(*SOA 12.01.2023 {  *)
(* QVis page 141, Warm up *)
iIndexPage:=141;
iPageNumber:=iPageNumber+1;
T_Visu.T_PageIndex[iIndexPage].iIndexConfigPage:=iPageNumber;
ptrConfigPage:=ADR(T_Visu.T_ConfigPage[T_Visu.T_PageIndex[iIndexPage].iIndexConfigPage]);
ptrConfigPage^.sName:='Warm up';
ptrConfigPage^.wMaskBtPanelLeft:=16#1F;
ptrConfigPage^.wMaskBtPanelRight:=16#60;
ptrConfigPage^.wMaskFunctionPanel:=16#31;
(* Navigation panel restriction *)
ptrConfigPage^.wMaskTouchScreenNavPanel:=16#3F;
(* Active machine movement mask *)
ptrConfigPage^.wMaskActiveMachineBtPanelLeft:=16#0;
ptrConfigPage^.wMaskActiveMachineBtPanelRight:=16#0;
ptrConfigPage^.wMaskActiveMachineFunctionPanel:=16#0;
ptrConfigPage^.wMaskActiveMachineNavPanel:=16#3F;
(* Button edge action *)
ptrConfigPage^.aiRTrigActionPanelRight[1]:=10140;
ptrConfigPage^.aiRTrigActionPanelRight[2]:=10141;
ptrConfigPage^.aiRTrigActionPanelRight[3]:=0;
ptrConfigPage^.aiRTrigActionPanelRight[4]:=0;
ptrConfigPage^.aiRTrigActionPanelRight[5]:=0;
ptrConfigPage^.aiFTrigActionPanelRight[1]:=0;
ptrConfigPage^.aiFTrigActionPanelRight[2]:=0;
ptrConfigPage^.aiFTrigActionPanelRight[3]:=0;
ptrConfigPage^.aiFTrigActionPanelRight[4]:=0;
ptrConfigPage^.aiFTrigActionPanelRight[5]:=0;
ptrConfigPage^.aiDelayActionPanelRight[1]:=0;
ptrConfigPage^.aiDelayActionPanelRight[2]:=0;
ptrConfigPage^.aiDelayActionPanelRight[3]:=0;
ptrConfigPage^.aiDelayActionPanelRight[4]:=0;
ptrConfigPage^.aiDelayActionPanelRight[5]:=0;
ptrConfigPage^.aiRTrigActionFunctionPanel[1]:=173;
ptrConfigPage^.aiRTrigActionFunctionPanel[2]:=0;
ptrConfigPage^.aiRTrigActionFunctionPanel[3]:=0;
ptrConfigPage^.aiRTrigActionFunctionPanel[4]:=0;
ptrConfigPage^.aiRTrigActionFunctionPanel[5]:=175;
ptrConfigPage^.aiRTrigActionFunctionPanel[6]:= 1005; (*Vorher: 171*)
ptrConfigPage^.aiRTrigActionFunctionPanel[7]:=0;
ptrConfigPage^.aiRTrigActionFunctionPanel[8]:=0;
ptrConfigPage^.aiRTrigActionFunctionPanel[9]:=0;
ptrConfigPage^.aiRTrigActionFunctionPanel[10]:=0;
ptrConfigPage^.aiRTrigActionFunctionPanel[11]:=0;
ptrConfigPage^.aiRTrigActionFunctionPanel[12]:=0;
ptrConfigPage^.aiFTrigActionTouchScreenNavPanel[1]:=10110;
ptrConfigPage^.aiFTrigActionTouchScreenNavPanel[2]:=10120;
ptrConfigPage^.aiFTrigActionTouchScreenNavPanel[3]:=10130;
ptrConfigPage^.aiFTrigActionTouchScreenNavPanel[4]:=10140;
ptrConfigPage^.aiFTrigActionTouchScreenNavPanel[5]:=10150;
ptrConfigPage^.aiFTrigActionTouchScreenNavPanel[6]:=10160;
ptrConfigPage^.xMaskBtStart:=FALSE;
ptrConfigPage^.xMaskBtStop:=TRUE;
(*SOA 12.01.2023 }  *)

(* QVis page 150, Configuration *)
iIndexPage:=150;
iPageNumber:=iPageNumber+1;
T_Visu.T_PageIndex[iIndexPage].iIndexConfigPage:=iPageNumber;
ptrConfigPage:=ADR(T_Visu.T_ConfigPage[T_Visu.T_PageIndex[iIndexPage].iIndexConfigPage]);
ptrConfigPage^.sName:='Configuration';
ptrConfigPage^.wMaskBtPanelLeft:=16#1F;
ptrConfigPage^.wMaskBtPanelRight:=16#0;
ptrConfigPage^.wMaskFunctionPanel:=16#0;
(* Navigation panel restriction *)
ptrConfigPage^.wMaskTouchScreenNavPanel:=16#3F;
(* Active machine movement mask *)
ptrConfigPage^.wMaskActiveMachineBtPanelLeft:=16#0;
ptrConfigPage^.wMaskActiveMachineBtPanelRight:=16#0;
ptrConfigPage^.wMaskActiveMachineFunctionPanel:=16#0;
ptrConfigPage^.wMaskActiveMachineNavPanel:=16#3F;
(* Button edge action *)
ptrConfigPage^.aiRTrigActionPanelRight[1]:=0;
ptrConfigPage^.aiRTrigActionPanelRight[2]:=0;
ptrConfigPage^.aiRTrigActionPanelRight[3]:=0;
ptrConfigPage^.aiRTrigActionPanelRight[4]:=0;
ptrConfigPage^.aiRTrigActionPanelRight[5]:=0;
ptrConfigPage^.aiFTrigActionPanelRight[1]:=0;
ptrConfigPage^.aiFTrigActionPanelRight[2]:=0;
ptrConfigPage^.aiFTrigActionPanelRight[3]:=0;
ptrConfigPage^.aiFTrigActionPanelRight[4]:=0;
ptrConfigPage^.aiFTrigActionPanelRight[5]:=0;
ptrConfigPage^.aiDelayActionPanelRight[1]:=0;
ptrConfigPage^.aiDelayActionPanelRight[2]:=0;
ptrConfigPage^.aiDelayActionPanelRight[3]:=0;
ptrConfigPage^.aiDelayActionPanelRight[4]:=0;
ptrConfigPage^.aiDelayActionPanelRight[5]:=0;
ptrConfigPage^.aiRTrigActionFunctionPanel[1]:=0;
ptrConfigPage^.aiRTrigActionFunctionPanel[2]:=0;
ptrConfigPage^.aiRTrigActionFunctionPanel[3]:=0;
ptrConfigPage^.aiRTrigActionFunctionPanel[4]:=0;
ptrConfigPage^.aiRTrigActionFunctionPanel[5]:=0;
ptrConfigPage^.aiRTrigActionFunctionPanel[6]:=0;
ptrConfigPage^.aiRTrigActionFunctionPanel[7]:=0;
ptrConfigPage^.aiRTrigActionFunctionPanel[8]:=0;
ptrConfigPage^.aiRTrigActionFunctionPanel[9]:=0;
ptrConfigPage^.aiRTrigActionFunctionPanel[10]:=0;
ptrConfigPage^.aiRTrigActionFunctionPanel[11]:=0;
ptrConfigPage^.aiRTrigActionFunctionPanel[12]:=0;
ptrConfigPage^.aiFTrigActionTouchScreenNavPanel[1]:=10110;
ptrConfigPage^.aiFTrigActionTouchScreenNavPanel[2]:=10120;
ptrConfigPage^.aiFTrigActionTouchScreenNavPanel[3]:=10130;
ptrConfigPage^.aiFTrigActionTouchScreenNavPanel[4]:=10140;
ptrConfigPage^.aiFTrigActionTouchScreenNavPanel[5]:=10150;
ptrConfigPage^.aiFTrigActionTouchScreenNavPanel[6]:=10160;
ptrConfigPage^.xMaskBtStart:=FALSE;
ptrConfigPage^.xMaskBtStop:=TRUE;

(* QVis page 160, Error List *)
iIndexPage:=160;
iPageNumber:=iPageNumber+1;
T_Visu.T_PageIndex[iIndexPage].iIndexConfigPage:=iPageNumber;
ptrConfigPage:=ADR(T_Visu.T_ConfigPage[T_Visu.T_PageIndex[iIndexPage].iIndexConfigPage]);
ptrConfigPage^.sName:='Error List';
ptrConfigPage^.wMaskBtPanelLeft:=16#1F;
ptrConfigPage^.wMaskBtPanelRight:=16#60;
ptrConfigPage^.wMaskFunctionPanel:=16#0;
(* Navigation panel restriction *)
ptrConfigPage^.wMaskTouchScreenNavPanel:=16#3F;
(* Active machine movement mask *)
ptrConfigPage^.wMaskActiveMachineBtPanelLeft:=16#0;
ptrConfigPage^.wMaskActiveMachineBtPanelRight:=16#60;
ptrConfigPage^.wMaskActiveMachineFunctionPanel:=16#0;
ptrConfigPage^.wMaskActiveMachineNavPanel:=16#3F;
(* Button edge action *)
ptrConfigPage^.aiRTrigActionPanelRight[1]:=99;
ptrConfigPage^.aiRTrigActionPanelRight[2]:=20;
ptrConfigPage^.aiRTrigActionPanelRight[3]:=0;
ptrConfigPage^.aiRTrigActionPanelRight[4]:=0;
ptrConfigPage^.aiRTrigActionPanelRight[5]:=0;
ptrConfigPage^.aiFTrigActionPanelRight[1]:=0;
ptrConfigPage^.aiFTrigActionPanelRight[2]:=0;
ptrConfigPage^.aiFTrigActionPanelRight[3]:=0;
ptrConfigPage^.aiFTrigActionPanelRight[4]:=0;
ptrConfigPage^.aiFTrigActionPanelRight[5]:=0;
ptrConfigPage^.aiDelayActionPanelRight[1]:=0;
ptrConfigPage^.aiDelayActionPanelRight[2]:=0;
ptrConfigPage^.aiDelayActionPanelRight[3]:=0;
ptrConfigPage^.aiDelayActionPanelRight[4]:=0;
ptrConfigPage^.aiDelayActionPanelRight[5]:=0;
ptrConfigPage^.aiRTrigActionFunctionPanel[1]:=0;
ptrConfigPage^.aiRTrigActionFunctionPanel[2]:=0;
ptrConfigPage^.aiRTrigActionFunctionPanel[3]:=0;
ptrConfigPage^.aiRTrigActionFunctionPanel[4]:=0;
ptrConfigPage^.aiRTrigActionFunctionPanel[5]:=0;
ptrConfigPage^.aiRTrigActionFunctionPanel[6]:=0;
ptrConfigPage^.aiRTrigActionFunctionPanel[7]:=0;
ptrConfigPage^.aiRTrigActionFunctionPanel[8]:=0;
ptrConfigPage^.aiRTrigActionFunctionPanel[9]:=0;
ptrConfigPage^.aiRTrigActionFunctionPanel[10]:=0;
ptrConfigPage^.aiRTrigActionFunctionPanel[11]:=0;
ptrConfigPage^.aiRTrigActionFunctionPanel[12]:=0;
ptrConfigPage^.aiFTrigActionTouchScreenNavPanel[1]:=10110;
ptrConfigPage^.aiFTrigActionTouchScreenNavPanel[2]:=10120;
ptrConfigPage^.aiFTrigActionTouchScreenNavPanel[3]:=10130;
ptrConfigPage^.aiFTrigActionTouchScreenNavPanel[4]:=10140;
ptrConfigPage^.aiFTrigActionTouchScreenNavPanel[5]:=10150;
ptrConfigPage^.aiFTrigActionTouchScreenNavPanel[6]:=10160;
ptrConfigPage^.xMaskBtStart:=FALSE;
ptrConfigPage^.xMaskBtStop:=TRUE;

(* QVis page 170, Parameter General *)
iIndexPage:=170;
iPageNumber:=iPageNumber+1;
T_Visu.T_PageIndex[iIndexPage].iIndexConfigPage:=iPageNumber;
ptrConfigPage:=ADR(T_Visu.T_ConfigPage[T_Visu.T_PageIndex[iIndexPage].iIndexConfigPage]);
ptrConfigPage^.sName:='Parameter General';
ptrConfigPage^.wMaskBtPanelLeft:=16#1F;
ptrConfigPage^.wMaskBtPanelRight:=16#200;
ptrConfigPage^.wMaskFunctionPanel:=16#0;
(* Navigation panel restriction *)
ptrConfigPage^.wMaskTouchScreenNavPanel:=16#3F;
(* Active machine movement mask *)
ptrConfigPage^.wMaskActiveMachineBtPanelLeft:=16#0;
ptrConfigPage^.wMaskActiveMachineBtPanelRight:=16#0;
ptrConfigPage^.wMaskActiveMachineFunctionPanel:=16#0;
ptrConfigPage^.wMaskActiveMachineNavPanel:=16#3F;
(* Button edge action *)
ptrConfigPage^.aiRTrigActionPanelRight[1]:=0;
ptrConfigPage^.aiRTrigActionPanelRight[2]:=0;
ptrConfigPage^.aiRTrigActionPanelRight[3]:=0;
ptrConfigPage^.aiRTrigActionPanelRight[4]:=0;
ptrConfigPage^.aiRTrigActionPanelRight[5]:=1006;
ptrConfigPage^.aiFTrigActionPanelRight[1]:=0;
ptrConfigPage^.aiFTrigActionPanelRight[2]:=0;
ptrConfigPage^.aiFTrigActionPanelRight[3]:=0;
ptrConfigPage^.aiFTrigActionPanelRight[4]:=0;
ptrConfigPage^.aiFTrigActionPanelRight[5]:=0;
ptrConfigPage^.aiDelayActionPanelRight[1]:=0;
ptrConfigPage^.aiDelayActionPanelRight[2]:=0;
ptrConfigPage^.aiDelayActionPanelRight[3]:=0;
ptrConfigPage^.aiDelayActionPanelRight[4]:=0;
ptrConfigPage^.aiDelayActionPanelRight[5]:=0;
ptrConfigPage^.aiRTrigActionFunctionPanel[1]:=0;
ptrConfigPage^.aiRTrigActionFunctionPanel[2]:=0;
ptrConfigPage^.aiRTrigActionFunctionPanel[3]:=0;
ptrConfigPage^.aiRTrigActionFunctionPanel[4]:=0;
ptrConfigPage^.aiRTrigActionFunctionPanel[5]:=0;
ptrConfigPage^.aiRTrigActionFunctionPanel[6]:=0;
ptrConfigPage^.aiRTrigActionFunctionPanel[7]:=0;
ptrConfigPage^.aiRTrigActionFunctionPanel[8]:=0;
ptrConfigPage^.aiRTrigActionFunctionPanel[9]:=0;
ptrConfigPage^.aiRTrigActionFunctionPanel[10]:=0;
ptrConfigPage^.aiRTrigActionFunctionPanel[11]:=0;
ptrConfigPage^.aiRTrigActionFunctionPanel[12]:=0;
ptrConfigPage^.aiFTrigActionTouchScreenNavPanel[1]:=10110;
ptrConfigPage^.aiFTrigActionTouchScreenNavPanel[2]:=10120;
ptrConfigPage^.aiFTrigActionTouchScreenNavPanel[3]:=10130;
ptrConfigPage^.aiFTrigActionTouchScreenNavPanel[4]:=10140;
ptrConfigPage^.aiFTrigActionTouchScreenNavPanel[5]:=10150;
ptrConfigPage^.aiFTrigActionTouchScreenNavPanel[6]:=10160;
ptrConfigPage^.xMaskBtStart:=FALSE;
ptrConfigPage^.xMaskBtStop:=TRUE;

(* QVis page 210, Teach-in Tool Rotation *)
iIndexPage:=210;
iPageNumber:=iPageNumber+1;
T_Visu.T_PageIndex[iIndexPage].iIndexConfigPage:=iPageNumber;
ptrConfigPage:=ADR(T_Visu.T_ConfigPage[T_Visu.T_PageIndex[iIndexPage].iIndexConfigPage]);
ptrConfigPage^.sName:='Teach-in Tool Rotation';
ptrConfigPage^.wMaskBtPanelLeft:=16#1F;
ptrConfigPage^.wMaskBtPanelRight:=16#1E0;
ptrConfigPage^.wMaskFunctionPanel:=16#F;
(* Navigation panel restriction *)
ptrConfigPage^.wMaskTouchScreenNavPanel:=16#27;
(* Active machine movement mask *)
ptrConfigPage^.wMaskActiveMachineBtPanelLeft:=16#0;
ptrConfigPage^.wMaskActiveMachineBtPanelRight:=16#0;
ptrConfigPage^.wMaskActiveMachineFunctionPanel:=16#0;
ptrConfigPage^.wMaskActiveMachineNavPanel:=16#27;
(* Button edge action *)
ptrConfigPage^.aiRTrigActionPanelRight[1]:=312;
ptrConfigPage^.aiRTrigActionPanelRight[2]:=310;
ptrConfigPage^.aiRTrigActionPanelRight[3]:=316;
ptrConfigPage^.aiRTrigActionPanelRight[4]:=314;
ptrConfigPage^.aiRTrigActionPanelRight[5]:=0;
ptrConfigPage^.aiFTrigActionPanelRight[1]:=0;
ptrConfigPage^.aiFTrigActionPanelRight[2]:=0;
ptrConfigPage^.aiFTrigActionPanelRight[3]:=301;
ptrConfigPage^.aiFTrigActionPanelRight[4]:=301;
ptrConfigPage^.aiFTrigActionPanelRight[5]:=0;
ptrConfigPage^.aiDelayActionPanelRight[1]:=0;
ptrConfigPage^.aiDelayActionPanelRight[2]:=0;
ptrConfigPage^.aiDelayActionPanelRight[3]:=0;
ptrConfigPage^.aiDelayActionPanelRight[4]:=0;
ptrConfigPage^.aiDelayActionPanelRight[5]:=0;
ptrConfigPage^.aiRTrigActionFunctionPanel[1]:=322;
ptrConfigPage^.aiRTrigActionFunctionPanel[2]:=323;
ptrConfigPage^.aiRTrigActionFunctionPanel[3]:=321;
ptrConfigPage^.aiRTrigActionFunctionPanel[4]:=320;
ptrConfigPage^.aiRTrigActionFunctionPanel[5]:=0;
ptrConfigPage^.aiRTrigActionFunctionPanel[6]:=0;
ptrConfigPage^.aiRTrigActionFunctionPanel[7]:=0;
ptrConfigPage^.aiRTrigActionFunctionPanel[8]:=0;
ptrConfigPage^.aiRTrigActionFunctionPanel[9]:=0;
ptrConfigPage^.aiRTrigActionFunctionPanel[10]:=0;
ptrConfigPage^.aiRTrigActionFunctionPanel[11]:=0;
ptrConfigPage^.aiRTrigActionFunctionPanel[12]:=0;
ptrConfigPage^.aiFTrigActionTouchScreenNavPanel[1]:=10210;
ptrConfigPage^.aiFTrigActionTouchScreenNavPanel[2]:=10220;
ptrConfigPage^.aiFTrigActionTouchScreenNavPanel[3]:=10230;
ptrConfigPage^.aiFTrigActionTouchScreenNavPanel[4]:=0;
ptrConfigPage^.aiFTrigActionTouchScreenNavPanel[5]:=0;
ptrConfigPage^.aiFTrigActionTouchScreenNavPanel[6]:=10260;
ptrConfigPage^.xMaskBtStart:=TRUE;
ptrConfigPage^.xMaskBtStop:=TRUE;

(* QVis page 220, Tool Torque *)
iIndexPage:=220;
iPageNumber:=iPageNumber+1;
T_Visu.T_PageIndex[iIndexPage].iIndexConfigPage:=iPageNumber;
ptrConfigPage:=ADR(T_Visu.T_ConfigPage[T_Visu.T_PageIndex[iIndexPage].iIndexConfigPage]);
ptrConfigPage^.sName:='Tool Torque';
ptrConfigPage^.wMaskBtPanelLeft:=16#1F;
ptrConfigPage^.wMaskBtPanelRight:=16#0;
ptrConfigPage^.wMaskFunctionPanel:=16#DF;
(* Navigation panel restriction *)
ptrConfigPage^.wMaskTouchScreenNavPanel:=16#27;
(* Active machine movement mask *)
ptrConfigPage^.wMaskActiveMachineBtPanelLeft:=16#0;
ptrConfigPage^.wMaskActiveMachineBtPanelRight:=16#0;
ptrConfigPage^.wMaskActiveMachineFunctionPanel:=16#DF;
ptrConfigPage^.wMaskActiveMachineNavPanel:=16#27;
(* Button edge action *)
ptrConfigPage^.aiRTrigActionPanelRight[1]:=0;
ptrConfigPage^.aiRTrigActionPanelRight[2]:=0;
ptrConfigPage^.aiRTrigActionPanelRight[3]:=0;
ptrConfigPage^.aiRTrigActionPanelRight[4]:=0;
ptrConfigPage^.aiRTrigActionPanelRight[5]:=0;
ptrConfigPage^.aiFTrigActionPanelRight[1]:=0;
ptrConfigPage^.aiFTrigActionPanelRight[2]:=0;
ptrConfigPage^.aiFTrigActionPanelRight[3]:=0;
ptrConfigPage^.aiFTrigActionPanelRight[4]:=0;
ptrConfigPage^.aiFTrigActionPanelRight[5]:=0;
ptrConfigPage^.aiDelayActionPanelRight[1]:=0;
ptrConfigPage^.aiDelayActionPanelRight[2]:=0;
ptrConfigPage^.aiDelayActionPanelRight[3]:=0;
ptrConfigPage^.aiDelayActionPanelRight[4]:=0;
ptrConfigPage^.aiDelayActionPanelRight[5]:=0;
ptrConfigPage^.aiRTrigActionFunctionPanel[1]:=502;
ptrConfigPage^.aiRTrigActionFunctionPanel[2]:=503;
ptrConfigPage^.aiRTrigActionFunctionPanel[3]:=501;
ptrConfigPage^.aiRTrigActionFunctionPanel[4]:=130;
ptrConfigPage^.aiRTrigActionFunctionPanel[5]:=131;
ptrConfigPage^.aiRTrigActionFunctionPanel[6]:=0;
ptrConfigPage^.aiRTrigActionFunctionPanel[7]:=504;
ptrConfigPage^.aiRTrigActionFunctionPanel[8]:=505;
ptrConfigPage^.aiRTrigActionFunctionPanel[9]:=0;
ptrConfigPage^.aiRTrigActionFunctionPanel[10]:=0;
ptrConfigPage^.aiRTrigActionFunctionPanel[11]:=0;
ptrConfigPage^.aiRTrigActionFunctionPanel[12]:=0;
ptrConfigPage^.aiFTrigActionTouchScreenNavPanel[1]:=10210;
ptrConfigPage^.aiFTrigActionTouchScreenNavPanel[2]:=10220;
ptrConfigPage^.aiFTrigActionTouchScreenNavPanel[3]:=10230;
ptrConfigPage^.aiFTrigActionTouchScreenNavPanel[4]:=0;
ptrConfigPage^.aiFTrigActionTouchScreenNavPanel[5]:=0;
ptrConfigPage^.aiFTrigActionTouchScreenNavPanel[6]:=10260;
ptrConfigPage^.xMaskBtStart:=TRUE;
ptrConfigPage^.xMaskBtStop:=TRUE;

(* QVis page 230, Tool Tension *)
iIndexPage:=230;
iPageNumber:=iPageNumber+1;
T_Visu.T_PageIndex[iIndexPage].iIndexConfigPage:=iPageNumber;
ptrConfigPage:=ADR(T_Visu.T_ConfigPage[T_Visu.T_PageIndex[iIndexPage].iIndexConfigPage]);
ptrConfigPage^.sName:='Tool Tension';
ptrConfigPage^.wMaskBtPanelLeft:=16#1F;
ptrConfigPage^.wMaskBtPanelRight:=16#20;
ptrConfigPage^.wMaskFunctionPanel:=16#0;
(* Navigation panel restriction *)
ptrConfigPage^.wMaskTouchScreenNavPanel:=16#27;
(* Active machine movement mask *)
ptrConfigPage^.wMaskActiveMachineBtPanelLeft:=16#0;
ptrConfigPage^.wMaskActiveMachineBtPanelRight:=16#0;
ptrConfigPage^.wMaskActiveMachineFunctionPanel:=16#0;
ptrConfigPage^.wMaskActiveMachineNavPanel:=16#27;
(* Button edge action *)
ptrConfigPage^.aiRTrigActionPanelRight[1]:=501;
ptrConfigPage^.aiRTrigActionPanelRight[2]:=0;
ptrConfigPage^.aiRTrigActionPanelRight[3]:=0;
ptrConfigPage^.aiRTrigActionPanelRight[4]:=0;
ptrConfigPage^.aiRTrigActionPanelRight[5]:=0;
ptrConfigPage^.aiFTrigActionPanelRight[1]:=0;
ptrConfigPage^.aiFTrigActionPanelRight[2]:=0;
ptrConfigPage^.aiFTrigActionPanelRight[3]:=0;
ptrConfigPage^.aiFTrigActionPanelRight[4]:=0;
ptrConfigPage^.aiFTrigActionPanelRight[5]:=0;
ptrConfigPage^.aiDelayActionPanelRight[1]:=0;
ptrConfigPage^.aiDelayActionPanelRight[2]:=0;
ptrConfigPage^.aiDelayActionPanelRight[3]:=0;
ptrConfigPage^.aiDelayActionPanelRight[4]:=0;
ptrConfigPage^.aiDelayActionPanelRight[5]:=0;
ptrConfigPage^.aiRTrigActionFunctionPanel[1]:=0;
ptrConfigPage^.aiRTrigActionFunctionPanel[2]:=0;
ptrConfigPage^.aiRTrigActionFunctionPanel[3]:=0;
ptrConfigPage^.aiRTrigActionFunctionPanel[4]:=0;
ptrConfigPage^.aiRTrigActionFunctionPanel[5]:=0;
ptrConfigPage^.aiRTrigActionFunctionPanel[6]:=0;
ptrConfigPage^.aiRTrigActionFunctionPanel[7]:=0;
ptrConfigPage^.aiRTrigActionFunctionPanel[8]:=0;
ptrConfigPage^.aiRTrigActionFunctionPanel[9]:=0;
ptrConfigPage^.aiRTrigActionFunctionPanel[10]:=0;
ptrConfigPage^.aiRTrigActionFunctionPanel[11]:=0;
ptrConfigPage^.aiRTrigActionFunctionPanel[12]:=0;
ptrConfigPage^.aiFTrigActionTouchScreenNavPanel[1]:=10210;
ptrConfigPage^.aiFTrigActionTouchScreenNavPanel[2]:=10220;
ptrConfigPage^.aiFTrigActionTouchScreenNavPanel[3]:=10230;
ptrConfigPage^.aiFTrigActionTouchScreenNavPanel[4]:=0;
ptrConfigPage^.aiFTrigActionTouchScreenNavPanel[5]:=0;
ptrConfigPage^.aiFTrigActionTouchScreenNavPanel[6]:=10260;
ptrConfigPage^.xMaskBtStart:=FALSE;
ptrConfigPage^.xMaskBtStop:=TRUE;

(* QVis page 260, Error List *)
iIndexPage:=260;
iPageNumber:=iPageNumber+1;
T_Visu.T_PageIndex[iIndexPage].iIndexConfigPage:=iPageNumber;
ptrConfigPage:=ADR(T_Visu.T_ConfigPage[T_Visu.T_PageIndex[iIndexPage].iIndexConfigPage]);
ptrConfigPage^.sName:='Error List';
ptrConfigPage^.wMaskBtPanelLeft:=16#1F;
ptrConfigPage^.wMaskBtPanelRight:=16#60;
ptrConfigPage^.wMaskFunctionPanel:=16#0;
(* Navigation panel restriction *)
ptrConfigPage^.wMaskTouchScreenNavPanel:=16#27;
(* Active machine movement mask *)
ptrConfigPage^.wMaskActiveMachineBtPanelLeft:=16#0;
ptrConfigPage^.wMaskActiveMachineBtPanelRight:=16#60;
ptrConfigPage^.wMaskActiveMachineFunctionPanel:=16#0;
ptrConfigPage^.wMaskActiveMachineNavPanel:=16#27;
(* Button edge action *)
ptrConfigPage^.aiRTrigActionPanelRight[1]:=99;
ptrConfigPage^.aiRTrigActionPanelRight[2]:=20;
ptrConfigPage^.aiRTrigActionPanelRight[3]:=0;
ptrConfigPage^.aiRTrigActionPanelRight[4]:=0;
ptrConfigPage^.aiRTrigActionPanelRight[5]:=0;
ptrConfigPage^.aiFTrigActionPanelRight[1]:=0;
ptrConfigPage^.aiFTrigActionPanelRight[2]:=0;
ptrConfigPage^.aiFTrigActionPanelRight[3]:=0;
ptrConfigPage^.aiFTrigActionPanelRight[4]:=0;
ptrConfigPage^.aiFTrigActionPanelRight[5]:=0;
ptrConfigPage^.aiDelayActionPanelRight[1]:=0;
ptrConfigPage^.aiDelayActionPanelRight[2]:=0;
ptrConfigPage^.aiDelayActionPanelRight[3]:=0;
ptrConfigPage^.aiDelayActionPanelRight[4]:=0;
ptrConfigPage^.aiDelayActionPanelRight[5]:=0;
ptrConfigPage^.aiRTrigActionFunctionPanel[1]:=0;
ptrConfigPage^.aiRTrigActionFunctionPanel[2]:=0;
ptrConfigPage^.aiRTrigActionFunctionPanel[3]:=0;
ptrConfigPage^.aiRTrigActionFunctionPanel[4]:=0;
ptrConfigPage^.aiRTrigActionFunctionPanel[5]:=0;
ptrConfigPage^.aiRTrigActionFunctionPanel[6]:=0;
ptrConfigPage^.aiRTrigActionFunctionPanel[7]:=0;
ptrConfigPage^.aiRTrigActionFunctionPanel[8]:=0;
ptrConfigPage^.aiRTrigActionFunctionPanel[9]:=0;
ptrConfigPage^.aiRTrigActionFunctionPanel[10]:=0;
ptrConfigPage^.aiRTrigActionFunctionPanel[11]:=0;
ptrConfigPage^.aiRTrigActionFunctionPanel[12]:=0;
ptrConfigPage^.aiFTrigActionTouchScreenNavPanel[1]:=10210;
ptrConfigPage^.aiFTrigActionTouchScreenNavPanel[2]:=10220;
ptrConfigPage^.aiFTrigActionTouchScreenNavPanel[3]:=10230;
ptrConfigPage^.aiFTrigActionTouchScreenNavPanel[4]:=0;
ptrConfigPage^.aiFTrigActionTouchScreenNavPanel[5]:=0;
ptrConfigPage^.aiFTrigActionTouchScreenNavPanel[6]:=10260;
ptrConfigPage^.xMaskBtStart:=FALSE;
ptrConfigPage^.xMaskBtStop:=TRUE;

(* QVis page 270, Parameter Tool Rotation *)
iIndexPage:=270;
iPageNumber:=iPageNumber+1;
T_Visu.T_PageIndex[iIndexPage].iIndexConfigPage:=iPageNumber;
ptrConfigPage:=ADR(T_Visu.T_ConfigPage[T_Visu.T_PageIndex[iIndexPage].iIndexConfigPage]);
ptrConfigPage^.sName:='Parameter Tool Rotation';
ptrConfigPage^.wMaskBtPanelLeft:=16#1F;
ptrConfigPage^.wMaskBtPanelRight:=16#200;
ptrConfigPage^.wMaskFunctionPanel:=16#0;
(* Navigation panel restriction *)
ptrConfigPage^.wMaskTouchScreenNavPanel:=16#27;
(* Active machine movement mask *)
ptrConfigPage^.wMaskActiveMachineBtPanelLeft:=16#0;
ptrConfigPage^.wMaskActiveMachineBtPanelRight:=16#0;
ptrConfigPage^.wMaskActiveMachineFunctionPanel:=16#0;
ptrConfigPage^.wMaskActiveMachineNavPanel:=16#27;
(* Button edge action *)
ptrConfigPage^.aiRTrigActionPanelRight[1]:=0;
ptrConfigPage^.aiRTrigActionPanelRight[2]:=0;
ptrConfigPage^.aiRTrigActionPanelRight[3]:=0;
ptrConfigPage^.aiRTrigActionPanelRight[4]:=0;
ptrConfigPage^.aiRTrigActionPanelRight[5]:=1006;
ptrConfigPage^.aiFTrigActionPanelRight[1]:=0;
ptrConfigPage^.aiFTrigActionPanelRight[2]:=0;
ptrConfigPage^.aiFTrigActionPanelRight[3]:=0;
ptrConfigPage^.aiFTrigActionPanelRight[4]:=0;
ptrConfigPage^.aiFTrigActionPanelRight[5]:=0;
ptrConfigPage^.aiDelayActionPanelRight[1]:=0;
ptrConfigPage^.aiDelayActionPanelRight[2]:=0;
ptrConfigPage^.aiDelayActionPanelRight[3]:=0;
ptrConfigPage^.aiDelayActionPanelRight[4]:=0;
ptrConfigPage^.aiDelayActionPanelRight[5]:=0;
ptrConfigPage^.aiRTrigActionFunctionPanel[1]:=0;
ptrConfigPage^.aiRTrigActionFunctionPanel[2]:=0;
ptrConfigPage^.aiRTrigActionFunctionPanel[3]:=0;
ptrConfigPage^.aiRTrigActionFunctionPanel[4]:=0;
ptrConfigPage^.aiRTrigActionFunctionPanel[5]:=0;
ptrConfigPage^.aiRTrigActionFunctionPanel[6]:=0;
ptrConfigPage^.aiRTrigActionFunctionPanel[7]:=0;
ptrConfigPage^.aiRTrigActionFunctionPanel[8]:=0;
ptrConfigPage^.aiRTrigActionFunctionPanel[9]:=0;
ptrConfigPage^.aiRTrigActionFunctionPanel[10]:=0;
ptrConfigPage^.aiRTrigActionFunctionPanel[11]:=0;
ptrConfigPage^.aiRTrigActionFunctionPanel[12]:=0;
ptrConfigPage^.aiFTrigActionTouchScreenNavPanel[1]:=10210;
ptrConfigPage^.aiFTrigActionTouchScreenNavPanel[2]:=10220;
ptrConfigPage^.aiFTrigActionTouchScreenNavPanel[3]:=10230;
ptrConfigPage^.aiFTrigActionTouchScreenNavPanel[4]:=0;
ptrConfigPage^.aiFTrigActionTouchScreenNavPanel[5]:=0;
ptrConfigPage^.aiFTrigActionTouchScreenNavPanel[6]:=10260;
ptrConfigPage^.xMaskBtStart:=FALSE;
ptrConfigPage^.xMaskBtStop:=TRUE;

(* QVis page 310, Teach-in Wire Feeder *)
iIndexPage:=310;
iPageNumber:=iPageNumber+1;
T_Visu.T_PageIndex[iIndexPage].iIndexConfigPage:=iPageNumber;
ptrConfigPage:=ADR(T_Visu.T_ConfigPage[T_Visu.T_PageIndex[iIndexPage].iIndexConfigPage]);
ptrConfigPage^.sName:='Teach-in Wire Feeder';
ptrConfigPage^.wMaskBtPanelLeft:=16#1F;
ptrConfigPage^.wMaskBtPanelRight:=16#1E0;
ptrConfigPage^.wMaskFunctionPanel:=16#3F;
(* Navigation panel restriction *)
ptrConfigPage^.wMaskTouchScreenNavPanel:=16#27;
(* Active machine movement mask *)
ptrConfigPage^.wMaskActiveMachineBtPanelLeft:=16#0;
ptrConfigPage^.wMaskActiveMachineBtPanelRight:=16#0;
ptrConfigPage^.wMaskActiveMachineFunctionPanel:=16#0;
ptrConfigPage^.wMaskActiveMachineNavPanel:=16#27;
(* Button edge action *)
ptrConfigPage^.aiRTrigActionPanelRight[1]:=312;
ptrConfigPage^.aiRTrigActionPanelRight[2]:=310;
ptrConfigPage^.aiRTrigActionPanelRight[3]:=316;
ptrConfigPage^.aiRTrigActionPanelRight[4]:=314;
ptrConfigPage^.aiRTrigActionPanelRight[5]:=0;
ptrConfigPage^.aiFTrigActionPanelRight[1]:=0;
ptrConfigPage^.aiFTrigActionPanelRight[2]:=0;
ptrConfigPage^.aiFTrigActionPanelRight[3]:=301;
ptrConfigPage^.aiFTrigActionPanelRight[4]:=301;
ptrConfigPage^.aiFTrigActionPanelRight[5]:=0;
ptrConfigPage^.aiDelayActionPanelRight[1]:=0;
ptrConfigPage^.aiDelayActionPanelRight[2]:=0;
ptrConfigPage^.aiDelayActionPanelRight[3]:=0;
ptrConfigPage^.aiDelayActionPanelRight[4]:=0;
ptrConfigPage^.aiDelayActionPanelRight[5]:=0;
ptrConfigPage^.aiRTrigActionFunctionPanel[1]:=322;
ptrConfigPage^.aiRTrigActionFunctionPanel[2]:=323;
ptrConfigPage^.aiRTrigActionFunctionPanel[3]:=324;
ptrConfigPage^.aiRTrigActionFunctionPanel[4]:=320;
ptrConfigPage^.aiRTrigActionFunctionPanel[5]:=501;
ptrConfigPage^.aiRTrigActionFunctionPanel[6]:=325;
ptrConfigPage^.aiRTrigActionFunctionPanel[7]:=0;
ptrConfigPage^.aiRTrigActionFunctionPanel[8]:=0;
ptrConfigPage^.aiRTrigActionFunctionPanel[9]:=0;
ptrConfigPage^.aiRTrigActionFunctionPanel[10]:=0;
ptrConfigPage^.aiRTrigActionFunctionPanel[11]:=0;
ptrConfigPage^.aiRTrigActionFunctionPanel[12]:=0;
ptrConfigPage^.aiFTrigActionTouchScreenNavPanel[1]:=10310;
ptrConfigPage^.aiFTrigActionTouchScreenNavPanel[2]:=10320;
ptrConfigPage^.aiFTrigActionTouchScreenNavPanel[3]:=10330;
ptrConfigPage^.aiFTrigActionTouchScreenNavPanel[4]:=0;
ptrConfigPage^.aiFTrigActionTouchScreenNavPanel[5]:=0;
ptrConfigPage^.aiFTrigActionTouchScreenNavPanel[6]:=10360;
ptrConfigPage^.xMaskBtStart:=TRUE;
ptrConfigPage^.xMaskBtStop:=TRUE;

(* QVis page 320, Setting-up *)
iIndexPage:=320;
iPageNumber:=iPageNumber+1;
T_Visu.T_PageIndex[iIndexPage].iIndexConfigPage:=iPageNumber;
ptrConfigPage:=ADR(T_Visu.T_ConfigPage[T_Visu.T_PageIndex[iIndexPage].iIndexConfigPage]);
ptrConfigPage^.sName:='Setting-up';
ptrConfigPage^.wMaskBtPanelLeft:=16#1F;
ptrConfigPage^.wMaskBtPanelRight:=16#60;
ptrConfigPage^.wMaskFunctionPanel:=16#F;
(* Navigation panel restriction *)
ptrConfigPage^.wMaskTouchScreenNavPanel:=16#27;
(* Active machine movement mask *)
ptrConfigPage^.wMaskActiveMachineBtPanelLeft:=16#0;
ptrConfigPage^.wMaskActiveMachineBtPanelRight:=16#0;
ptrConfigPage^.wMaskActiveMachineFunctionPanel:=16#0;
ptrConfigPage^.wMaskActiveMachineNavPanel:=16#27;
(* Button edge action *)
ptrConfigPage^.aiRTrigActionPanelRight[1]:=312;
ptrConfigPage^.aiRTrigActionPanelRight[2]:=310;
ptrConfigPage^.aiRTrigActionPanelRight[3]:=0;
ptrConfigPage^.aiRTrigActionPanelRight[4]:=0;
ptrConfigPage^.aiRTrigActionPanelRight[5]:=0;
ptrConfigPage^.aiFTrigActionPanelRight[1]:=301;
ptrConfigPage^.aiFTrigActionPanelRight[2]:=301;
ptrConfigPage^.aiFTrigActionPanelRight[3]:=0;
ptrConfigPage^.aiFTrigActionPanelRight[4]:=0;
ptrConfigPage^.aiFTrigActionPanelRight[5]:=0;
ptrConfigPage^.aiDelayActionPanelRight[1]:=316;
ptrConfigPage^.aiDelayActionPanelRight[2]:=314;
ptrConfigPage^.aiDelayActionPanelRight[3]:=0;
ptrConfigPage^.aiDelayActionPanelRight[4]:=0;
ptrConfigPage^.aiDelayActionPanelRight[5]:=0;
ptrConfigPage^.aiRTrigActionFunctionPanel[1]:=322;
ptrConfigPage^.aiRTrigActionFunctionPanel[2]:=323;
ptrConfigPage^.aiRTrigActionFunctionPanel[3]:=326;
ptrConfigPage^.aiRTrigActionFunctionPanel[4]:=320;
ptrConfigPage^.aiRTrigActionFunctionPanel[5]:=0;
ptrConfigPage^.aiRTrigActionFunctionPanel[6]:=0;
ptrConfigPage^.aiRTrigActionFunctionPanel[7]:=0;
ptrConfigPage^.aiRTrigActionFunctionPanel[8]:=0;
ptrConfigPage^.aiRTrigActionFunctionPanel[9]:=0;
ptrConfigPage^.aiRTrigActionFunctionPanel[10]:=0;
ptrConfigPage^.aiRTrigActionFunctionPanel[11]:=0;
ptrConfigPage^.aiRTrigActionFunctionPanel[12]:=0;
ptrConfigPage^.aiFTrigActionTouchScreenNavPanel[1]:=10310;
ptrConfigPage^.aiFTrigActionTouchScreenNavPanel[2]:=10320;
ptrConfigPage^.aiFTrigActionTouchScreenNavPanel[3]:=10330;
ptrConfigPage^.aiFTrigActionTouchScreenNavPanel[4]:=0;
ptrConfigPage^.aiFTrigActionTouchScreenNavPanel[5]:=0;
ptrConfigPage^.aiFTrigActionTouchScreenNavPanel[6]:=10360;
ptrConfigPage^.xMaskBtStart:=FALSE;
ptrConfigPage^.xMaskBtStop:=TRUE;

(* QVis page 330, ReferenceMaxToolLength *)
iIndexPage:=330;
iPageNumber:=iPageNumber+1;
T_Visu.T_PageIndex[iIndexPage].iIndexConfigPage:=iPageNumber;
ptrConfigPage:=ADR(T_Visu.T_ConfigPage[T_Visu.T_PageIndex[iIndexPage].iIndexConfigPage]);
ptrConfigPage^.sName:='Reference max ToolLength';
ptrConfigPage^.wMaskBtPanelLeft:=16#1F;
ptrConfigPage^.wMaskBtPanelRight:=16#1E0;
ptrConfigPage^.wMaskFunctionPanel:=16#1B;
(* Navigation panel restriction *)
ptrConfigPage^.wMaskTouchScreenNavPanel:=16#27;
(* Active machine movement mask *)
ptrConfigPage^.wMaskActiveMachineBtPanelLeft:=16#0;
ptrConfigPage^.wMaskActiveMachineBtPanelRight:=16#0;
ptrConfigPage^.wMaskActiveMachineFunctionPanel:=16#0;
ptrConfigPage^.wMaskActiveMachineNavPanel:=16#27;
(* Button edge action *)
ptrConfigPage^.aiRTrigActionPanelRight[1]:=312;
ptrConfigPage^.aiRTrigActionPanelRight[2]:=310;
ptrConfigPage^.aiRTrigActionPanelRight[3]:=316;
ptrConfigPage^.aiRTrigActionPanelRight[4]:=314;
ptrConfigPage^.aiRTrigActionPanelRight[5]:=0;
ptrConfigPage^.aiFTrigActionPanelRight[1]:=0;
ptrConfigPage^.aiFTrigActionPanelRight[2]:=0;
ptrConfigPage^.aiFTrigActionPanelRight[3]:=301;
ptrConfigPage^.aiFTrigActionPanelRight[4]:=301;
ptrConfigPage^.aiFTrigActionPanelRight[5]:=0;
ptrConfigPage^.aiDelayActionPanelRight[1]:=0;
ptrConfigPage^.aiDelayActionPanelRight[2]:=0;
ptrConfigPage^.aiDelayActionPanelRight[3]:=0;
ptrConfigPage^.aiDelayActionPanelRight[4]:=0;
ptrConfigPage^.aiDelayActionPanelRight[5]:=0;
ptrConfigPage^.aiRTrigActionFunctionPanel[1]:=322;
ptrConfigPage^.aiRTrigActionFunctionPanel[2]:=323;
ptrConfigPage^.aiRTrigActionFunctionPanel[3]:=0;
ptrConfigPage^.aiRTrigActionFunctionPanel[4]:=320;
ptrConfigPage^.aiRTrigActionFunctionPanel[5]:=501;
ptrConfigPage^.aiRTrigActionFunctionPanel[6]:=0;
ptrConfigPage^.aiRTrigActionFunctionPanel[7]:=0;
ptrConfigPage^.aiRTrigActionFunctionPanel[8]:=0;
ptrConfigPage^.aiRTrigActionFunctionPanel[9]:=0;
ptrConfigPage^.aiRTrigActionFunctionPanel[10]:=0;
ptrConfigPage^.aiRTrigActionFunctionPanel[11]:=0;
ptrConfigPage^.aiRTrigActionFunctionPanel[12]:=0;
ptrConfigPage^.aiFTrigActionTouchScreenNavPanel[1]:=10310;
ptrConfigPage^.aiFTrigActionTouchScreenNavPanel[2]:=10320;
ptrConfigPage^.aiFTrigActionTouchScreenNavPanel[3]:=10330;
ptrConfigPage^.aiFTrigActionTouchScreenNavPanel[4]:=0;
ptrConfigPage^.aiFTrigActionTouchScreenNavPanel[5]:=0;
ptrConfigPage^.aiFTrigActionTouchScreenNavPanel[6]:=10360;
ptrConfigPage^.xMaskBtStart:=TRUE;
ptrConfigPage^.xMaskBtStop:=TRUE;

(* QVis page 360, Error List *)
iIndexPage:=360;
iPageNumber:=iPageNumber+1;
T_Visu.T_PageIndex[iIndexPage].iIndexConfigPage:=iPageNumber;
ptrConfigPage:=ADR(T_Visu.T_ConfigPage[T_Visu.T_PageIndex[iIndexPage].iIndexConfigPage]);
ptrConfigPage^.sName:='Error List';
ptrConfigPage^.wMaskBtPanelLeft:=16#1F;
ptrConfigPage^.wMaskBtPanelRight:=16#60;
ptrConfigPage^.wMaskFunctionPanel:=16#0;
(* Navigation panel restriction *)
ptrConfigPage^.wMaskTouchScreenNavPanel:=16#27;
(* Active machine movement mask *)
ptrConfigPage^.wMaskActiveMachineBtPanelLeft:=16#0;
ptrConfigPage^.wMaskActiveMachineBtPanelRight:=16#60;
ptrConfigPage^.wMaskActiveMachineFunctionPanel:=16#0;
ptrConfigPage^.wMaskActiveMachineNavPanel:=16#27;
(* Button edge action *)
ptrConfigPage^.aiRTrigActionPanelRight[1]:=99;
ptrConfigPage^.aiRTrigActionPanelRight[2]:=20;
ptrConfigPage^.aiRTrigActionPanelRight[3]:=0;
ptrConfigPage^.aiRTrigActionPanelRight[4]:=0;
ptrConfigPage^.aiRTrigActionPanelRight[5]:=0;
ptrConfigPage^.aiFTrigActionPanelRight[1]:=0;
ptrConfigPage^.aiFTrigActionPanelRight[2]:=0;
ptrConfigPage^.aiFTrigActionPanelRight[3]:=0;
ptrConfigPage^.aiFTrigActionPanelRight[4]:=0;
ptrConfigPage^.aiFTrigActionPanelRight[5]:=0;
ptrConfigPage^.aiDelayActionPanelRight[1]:=0;
ptrConfigPage^.aiDelayActionPanelRight[2]:=0;
ptrConfigPage^.aiDelayActionPanelRight[3]:=0;
ptrConfigPage^.aiDelayActionPanelRight[4]:=0;
ptrConfigPage^.aiDelayActionPanelRight[5]:=0;
ptrConfigPage^.aiRTrigActionFunctionPanel[1]:=0;
ptrConfigPage^.aiRTrigActionFunctionPanel[2]:=0;
ptrConfigPage^.aiRTrigActionFunctionPanel[3]:=0;
ptrConfigPage^.aiRTrigActionFunctionPanel[4]:=0;
ptrConfigPage^.aiRTrigActionFunctionPanel[5]:=0;
ptrConfigPage^.aiRTrigActionFunctionPanel[6]:=0;
ptrConfigPage^.aiRTrigActionFunctionPanel[7]:=0;
ptrConfigPage^.aiRTrigActionFunctionPanel[8]:=0;
ptrConfigPage^.aiRTrigActionFunctionPanel[9]:=0;
ptrConfigPage^.aiRTrigActionFunctionPanel[10]:=0;
ptrConfigPage^.aiRTrigActionFunctionPanel[11]:=0;
ptrConfigPage^.aiRTrigActionFunctionPanel[12]:=0;
ptrConfigPage^.aiFTrigActionTouchScreenNavPanel[1]:=10310;
ptrConfigPage^.aiFTrigActionTouchScreenNavPanel[2]:=10320;
ptrConfigPage^.aiFTrigActionTouchScreenNavPanel[3]:=10330;
ptrConfigPage^.aiFTrigActionTouchScreenNavPanel[4]:=0;
ptrConfigPage^.aiFTrigActionTouchScreenNavPanel[5]:=0;
ptrConfigPage^.aiFTrigActionTouchScreenNavPanel[6]:=10360;
ptrConfigPage^.xMaskBtStart:=FALSE;
ptrConfigPage^.xMaskBtStop:=TRUE;

(* QVis page 370, Parameter Wire Feeder *)
iIndexPage:=370;
iPageNumber:=iPageNumber+1;
T_Visu.T_PageIndex[iIndexPage].iIndexConfigPage:=iPageNumber;
ptrConfigPage:=ADR(T_Visu.T_ConfigPage[T_Visu.T_PageIndex[iIndexPage].iIndexConfigPage]);
ptrConfigPage^.sName:='Parameter Wire Feeder';
ptrConfigPage^.wMaskBtPanelLeft:=16#1F;
ptrConfigPage^.wMaskBtPanelRight:=16#200;
ptrConfigPage^.wMaskFunctionPanel:=16#0;
(* Navigation panel restriction *)
ptrConfigPage^.wMaskTouchScreenNavPanel:=16#27;
(* Active machine movement mask *)
ptrConfigPage^.wMaskActiveMachineBtPanelLeft:=16#0;
ptrConfigPage^.wMaskActiveMachineBtPanelRight:=16#0;
ptrConfigPage^.wMaskActiveMachineFunctionPanel:=16#0;
ptrConfigPage^.wMaskActiveMachineNavPanel:=16#27;
(* Button edge action *)
ptrConfigPage^.aiRTrigActionPanelRight[1]:=0;
ptrConfigPage^.aiRTrigActionPanelRight[2]:=0;
ptrConfigPage^.aiRTrigActionPanelRight[3]:=0;
ptrConfigPage^.aiRTrigActionPanelRight[4]:=0;
ptrConfigPage^.aiRTrigActionPanelRight[5]:=1006;
ptrConfigPage^.aiFTrigActionPanelRight[1]:=0;
ptrConfigPage^.aiFTrigActionPanelRight[2]:=0;
ptrConfigPage^.aiFTrigActionPanelRight[3]:=0;
ptrConfigPage^.aiFTrigActionPanelRight[4]:=0;
ptrConfigPage^.aiFTrigActionPanelRight[5]:=0;
ptrConfigPage^.aiDelayActionPanelRight[1]:=0;
ptrConfigPage^.aiDelayActionPanelRight[2]:=0;
ptrConfigPage^.aiDelayActionPanelRight[3]:=0;
ptrConfigPage^.aiDelayActionPanelRight[4]:=0;
ptrConfigPage^.aiDelayActionPanelRight[5]:=0;
ptrConfigPage^.aiRTrigActionFunctionPanel[1]:=0;
ptrConfigPage^.aiRTrigActionFunctionPanel[2]:=0;
ptrConfigPage^.aiRTrigActionFunctionPanel[3]:=0;
ptrConfigPage^.aiRTrigActionFunctionPanel[4]:=0;
ptrConfigPage^.aiRTrigActionFunctionPanel[5]:=0;
ptrConfigPage^.aiRTrigActionFunctionPanel[6]:=0;
ptrConfigPage^.aiRTrigActionFunctionPanel[7]:=0;
ptrConfigPage^.aiRTrigActionFunctionPanel[8]:=0;
ptrConfigPage^.aiRTrigActionFunctionPanel[9]:=0;
ptrConfigPage^.aiRTrigActionFunctionPanel[10]:=0;
ptrConfigPage^.aiRTrigActionFunctionPanel[11]:=0;
ptrConfigPage^.aiRTrigActionFunctionPanel[12]:=0;
ptrConfigPage^.aiFTrigActionTouchScreenNavPanel[1]:=10310;
ptrConfigPage^.aiFTrigActionTouchScreenNavPanel[2]:=10320;
ptrConfigPage^.aiFTrigActionTouchScreenNavPanel[3]:=10330;
ptrConfigPage^.aiFTrigActionTouchScreenNavPanel[4]:=0;
ptrConfigPage^.aiFTrigActionTouchScreenNavPanel[5]:=0;
ptrConfigPage^.aiFTrigActionTouchScreenNavPanel[6]:=10360;
ptrConfigPage^.xMaskBtStart:=FALSE;
ptrConfigPage^.xMaskBtStop:=TRUE;

(* QVis page 410, Teach-in Grind Axis *)
iIndexPage:=410;
iPageNumber:=iPageNumber+1;
T_Visu.T_PageIndex[iIndexPage].iIndexConfigPage:=iPageNumber;
ptrConfigPage:=ADR(T_Visu.T_ConfigPage[T_Visu.T_PageIndex[iIndexPage].iIndexConfigPage]);
ptrConfigPage^.sName:='Teach-in Grind Axis';
ptrConfigPage^.wMaskBtPanelLeft:=16#1F;
ptrConfigPage^.wMaskBtPanelRight:=16#1E0;
ptrConfigPage^.wMaskFunctionPanel:=16#2B;
(* Navigation panel restriction *)
ptrConfigPage^.wMaskTouchScreenNavPanel:=16#27;
(* Active machine movement mask *)
ptrConfigPage^.wMaskActiveMachineBtPanelLeft:=16#0;
ptrConfigPage^.wMaskActiveMachineBtPanelRight:=16#0;
ptrConfigPage^.wMaskActiveMachineFunctionPanel:=16#0;
ptrConfigPage^.wMaskActiveMachineNavPanel:=16#27;
(* Button edge action *)
ptrConfigPage^.aiRTrigActionPanelRight[1]:=312;
ptrConfigPage^.aiRTrigActionPanelRight[2]:=310;
ptrConfigPage^.aiRTrigActionPanelRight[3]:=316;
ptrConfigPage^.aiRTrigActionPanelRight[4]:=314;
ptrConfigPage^.aiRTrigActionPanelRight[5]:=0;
ptrConfigPage^.aiFTrigActionPanelRight[1]:=0;
ptrConfigPage^.aiFTrigActionPanelRight[2]:=0;
ptrConfigPage^.aiFTrigActionPanelRight[3]:=301;
ptrConfigPage^.aiFTrigActionPanelRight[4]:=301;
ptrConfigPage^.aiFTrigActionPanelRight[5]:=0;
ptrConfigPage^.aiDelayActionPanelRight[1]:=0;
ptrConfigPage^.aiDelayActionPanelRight[2]:=0;
ptrConfigPage^.aiDelayActionPanelRight[3]:=0;
ptrConfigPage^.aiDelayActionPanelRight[4]:=0;
ptrConfigPage^.aiDelayActionPanelRight[5]:=0;
ptrConfigPage^.aiRTrigActionFunctionPanel[1]:=322;
ptrConfigPage^.aiRTrigActionFunctionPanel[2]:=323;
ptrConfigPage^.aiRTrigActionFunctionPanel[3]:=0;
ptrConfigPage^.aiRTrigActionFunctionPanel[4]:=320;
ptrConfigPage^.aiRTrigActionFunctionPanel[5]:=0;
ptrConfigPage^.aiRTrigActionFunctionPanel[6]:=325;
ptrConfigPage^.aiRTrigActionFunctionPanel[7]:=0;
ptrConfigPage^.aiRTrigActionFunctionPanel[8]:=0;
ptrConfigPage^.aiRTrigActionFunctionPanel[9]:=0;
ptrConfigPage^.aiRTrigActionFunctionPanel[10]:=0;
ptrConfigPage^.aiRTrigActionFunctionPanel[11]:=0;
ptrConfigPage^.aiRTrigActionFunctionPanel[12]:=0;
ptrConfigPage^.aiFTrigActionTouchScreenNavPanel[1]:=10410;
ptrConfigPage^.aiFTrigActionTouchScreenNavPanel[2]:=10420;
ptrConfigPage^.aiFTrigActionTouchScreenNavPanel[3]:=10430;
ptrConfigPage^.aiFTrigActionTouchScreenNavPanel[4]:=0;
ptrConfigPage^.aiFTrigActionTouchScreenNavPanel[5]:=0;
ptrConfigPage^.aiFTrigActionTouchScreenNavPanel[6]:=10460;
ptrConfigPage^.xMaskBtStart:=TRUE;
ptrConfigPage^.xMaskBtStop:=TRUE;

(* QVis page 420, Tool Diameter *)
iIndexPage:=420;
iPageNumber:=iPageNumber+1;
T_Visu.T_PageIndex[iIndexPage].iIndexConfigPage:=iPageNumber;
ptrConfigPage:=ADR(T_Visu.T_ConfigPage[T_Visu.T_PageIndex[iIndexPage].iIndexConfigPage]);
ptrConfigPage^.sName:='Tool Diameter';
ptrConfigPage^.wMaskBtPanelLeft:=16#1F;
ptrConfigPage^.wMaskBtPanelRight:=16#0;
ptrConfigPage^.wMaskFunctionPanel:=16#EF;
(* Navigation panel restriction *)
ptrConfigPage^.wMaskTouchScreenNavPanel:=16#27;
(* Active machine movement mask *)
ptrConfigPage^.wMaskActiveMachineBtPanelLeft:=16#0;
ptrConfigPage^.wMaskActiveMachineBtPanelRight:=16#0;
ptrConfigPage^.wMaskActiveMachineFunctionPanel:=16#0;
ptrConfigPage^.wMaskActiveMachineNavPanel:=16#27;
(* Button edge action *)
ptrConfigPage^.aiRTrigActionPanelRight[1]:=0;
ptrConfigPage^.aiRTrigActionPanelRight[2]:=0;
ptrConfigPage^.aiRTrigActionPanelRight[3]:=0;
ptrConfigPage^.aiRTrigActionPanelRight[4]:=0;
ptrConfigPage^.aiRTrigActionPanelRight[5]:=0;
ptrConfigPage^.aiFTrigActionPanelRight[1]:=0;
ptrConfigPage^.aiFTrigActionPanelRight[2]:=0;
ptrConfigPage^.aiFTrigActionPanelRight[3]:=0;
ptrConfigPage^.aiFTrigActionPanelRight[4]:=0;
ptrConfigPage^.aiFTrigActionPanelRight[5]:=0;
ptrConfigPage^.aiDelayActionPanelRight[1]:=0;
ptrConfigPage^.aiDelayActionPanelRight[2]:=0;
ptrConfigPage^.aiDelayActionPanelRight[3]:=0;
ptrConfigPage^.aiDelayActionPanelRight[4]:=0;
ptrConfigPage^.aiDelayActionPanelRight[5]:=0;
ptrConfigPage^.aiRTrigActionFunctionPanel[1]:=110;
ptrConfigPage^.aiRTrigActionFunctionPanel[2]:=111;
ptrConfigPage^.aiRTrigActionFunctionPanel[3]:=114;
ptrConfigPage^.aiRTrigActionFunctionPanel[4]:=115;
ptrConfigPage^.aiRTrigActionFunctionPanel[5]:=0;
ptrConfigPage^.aiRTrigActionFunctionPanel[6]:=116;
ptrConfigPage^.aiRTrigActionFunctionPanel[7]:=112;
ptrConfigPage^.aiRTrigActionFunctionPanel[8]:=113;
ptrConfigPage^.aiRTrigActionFunctionPanel[9]:=0;
ptrConfigPage^.aiRTrigActionFunctionPanel[10]:=0;
ptrConfigPage^.aiRTrigActionFunctionPanel[11]:=0;
ptrConfigPage^.aiRTrigActionFunctionPanel[12]:=0;
ptrConfigPage^.aiFTrigActionTouchScreenNavPanel[1]:=10410;
ptrConfigPage^.aiFTrigActionTouchScreenNavPanel[2]:=10420;
ptrConfigPage^.aiFTrigActionTouchScreenNavPanel[3]:=10430;
ptrConfigPage^.aiFTrigActionTouchScreenNavPanel[4]:=0;
ptrConfigPage^.aiFTrigActionTouchScreenNavPanel[5]:=0;
ptrConfigPage^.aiFTrigActionTouchScreenNavPanel[6]:=10460;
ptrConfigPage^.xMaskBtStart:=FALSE;
ptrConfigPage^.xMaskBtStop:=TRUE;

(* QVis page 430, Prism *)
iIndexPage:=430;
iPageNumber:=iPageNumber+1;
T_Visu.T_PageIndex[iIndexPage].iIndexConfigPage:=iPageNumber;
ptrConfigPage:=ADR(T_Visu.T_ConfigPage[T_Visu.T_PageIndex[iIndexPage].iIndexConfigPage]);
ptrConfigPage^.sName:='Prism';
ptrConfigPage^.wMaskBtPanelLeft:=16#1F;
ptrConfigPage^.wMaskBtPanelRight:=16#0;
ptrConfigPage^.wMaskFunctionPanel:=16#3F;
(* Navigation panel restriction *)
ptrConfigPage^.wMaskTouchScreenNavPanel:=16#27;
(* Active machine movement mask *)
ptrConfigPage^.wMaskActiveMachineBtPanelLeft:=16#0;
ptrConfigPage^.wMaskActiveMachineBtPanelRight:=16#0;
ptrConfigPage^.wMaskActiveMachineFunctionPanel:=16#0;
ptrConfigPage^.wMaskActiveMachineNavPanel:=16#27;
(* Button edge action *)
ptrConfigPage^.aiRTrigActionPanelRight[1]:=0;
ptrConfigPage^.aiRTrigActionPanelRight[2]:=0;
ptrConfigPage^.aiRTrigActionPanelRight[3]:=0;
ptrConfigPage^.aiRTrigActionPanelRight[4]:=0;
ptrConfigPage^.aiRTrigActionPanelRight[5]:=0;
ptrConfigPage^.aiFTrigActionPanelRight[1]:=0;
ptrConfigPage^.aiFTrigActionPanelRight[2]:=0;
ptrConfigPage^.aiFTrigActionPanelRight[3]:=0;
ptrConfigPage^.aiFTrigActionPanelRight[4]:=0;
ptrConfigPage^.aiFTrigActionPanelRight[5]:=0;
ptrConfigPage^.aiDelayActionPanelRight[1]:=0;
ptrConfigPage^.aiDelayActionPanelRight[2]:=0;
ptrConfigPage^.aiDelayActionPanelRight[3]:=0;
ptrConfigPage^.aiDelayActionPanelRight[4]:=0;
ptrConfigPage^.aiDelayActionPanelRight[5]:=0;
ptrConfigPage^.aiRTrigActionFunctionPanel[1]:=120;
ptrConfigPage^.aiRTrigActionFunctionPanel[2]:=115;
ptrConfigPage^.aiRTrigActionFunctionPanel[3]:=0;
ptrConfigPage^.aiRTrigActionFunctionPanel[4]:=0;
ptrConfigPage^.aiRTrigActionFunctionPanel[5]:=0;
ptrConfigPage^.aiRTrigActionFunctionPanel[6]:=1005;
ptrConfigPage^.aiRTrigActionFunctionPanel[7]:=0;
ptrConfigPage^.aiRTrigActionFunctionPanel[8]:=0;
ptrConfigPage^.aiRTrigActionFunctionPanel[9]:=0;
ptrConfigPage^.aiRTrigActionFunctionPanel[10]:=0;
ptrConfigPage^.aiRTrigActionFunctionPanel[11]:=0;
ptrConfigPage^.aiRTrigActionFunctionPanel[12]:=0;
ptrConfigPage^.aiFTrigActionTouchScreenNavPanel[1]:=10410;
ptrConfigPage^.aiFTrigActionTouchScreenNavPanel[2]:=10420;
ptrConfigPage^.aiFTrigActionTouchScreenNavPanel[3]:=10430;
ptrConfigPage^.aiFTrigActionTouchScreenNavPanel[4]:=0;
ptrConfigPage^.aiFTrigActionTouchScreenNavPanel[5]:=0;
ptrConfigPage^.aiFTrigActionTouchScreenNavPanel[6]:=10460;
ptrConfigPage^.xMaskBtStart:=FALSE;
ptrConfigPage^.xMaskBtStop:=TRUE;

(* QVis page 460, Error List *)
iIndexPage:=460;
iPageNumber:=iPageNumber+1;
T_Visu.T_PageIndex[iIndexPage].iIndexConfigPage:=iPageNumber;
ptrConfigPage:=ADR(T_Visu.T_ConfigPage[T_Visu.T_PageIndex[iIndexPage].iIndexConfigPage]);
ptrConfigPage^.sName:='Error List';
ptrConfigPage^.wMaskBtPanelLeft:=16#1F;
ptrConfigPage^.wMaskBtPanelRight:=16#60;
ptrConfigPage^.wMaskFunctionPanel:=16#0;
(* Navigation panel restriction *)
ptrConfigPage^.wMaskTouchScreenNavPanel:=16#27;
(* Active machine movement mask *)
ptrConfigPage^.wMaskActiveMachineBtPanelLeft:=16#0;
ptrConfigPage^.wMaskActiveMachineBtPanelRight:=16#60;
ptrConfigPage^.wMaskActiveMachineFunctionPanel:=16#0;
ptrConfigPage^.wMaskActiveMachineNavPanel:=16#27;
(* Button edge action *)
ptrConfigPage^.aiRTrigActionPanelRight[1]:=99;
ptrConfigPage^.aiRTrigActionPanelRight[2]:=20;
ptrConfigPage^.aiRTrigActionPanelRight[3]:=0;
ptrConfigPage^.aiRTrigActionPanelRight[4]:=0;
ptrConfigPage^.aiRTrigActionPanelRight[5]:=0;
ptrConfigPage^.aiFTrigActionPanelRight[1]:=0;
ptrConfigPage^.aiFTrigActionPanelRight[2]:=0;
ptrConfigPage^.aiFTrigActionPanelRight[3]:=0;
ptrConfigPage^.aiFTrigActionPanelRight[4]:=0;
ptrConfigPage^.aiFTrigActionPanelRight[5]:=0;
ptrConfigPage^.aiDelayActionPanelRight[1]:=0;
ptrConfigPage^.aiDelayActionPanelRight[2]:=0;
ptrConfigPage^.aiDelayActionPanelRight[3]:=0;
ptrConfigPage^.aiDelayActionPanelRight[4]:=0;
ptrConfigPage^.aiDelayActionPanelRight[5]:=0;
ptrConfigPage^.aiRTrigActionFunctionPanel[1]:=0;
ptrConfigPage^.aiRTrigActionFunctionPanel[2]:=0;
ptrConfigPage^.aiRTrigActionFunctionPanel[3]:=0;
ptrConfigPage^.aiRTrigActionFunctionPanel[4]:=0;
ptrConfigPage^.aiRTrigActionFunctionPanel[5]:=0;
ptrConfigPage^.aiRTrigActionFunctionPanel[6]:=0;
ptrConfigPage^.aiRTrigActionFunctionPanel[7]:=0;
ptrConfigPage^.aiRTrigActionFunctionPanel[8]:=0;
ptrConfigPage^.aiRTrigActionFunctionPanel[9]:=0;
ptrConfigPage^.aiRTrigActionFunctionPanel[10]:=0;
ptrConfigPage^.aiRTrigActionFunctionPanel[11]:=0;
ptrConfigPage^.aiRTrigActionFunctionPanel[12]:=0;
ptrConfigPage^.aiFTrigActionTouchScreenNavPanel[1]:=10410;
ptrConfigPage^.aiFTrigActionTouchScreenNavPanel[2]:=10420;
ptrConfigPage^.aiFTrigActionTouchScreenNavPanel[3]:=10430;
ptrConfigPage^.aiFTrigActionTouchScreenNavPanel[4]:=0;
ptrConfigPage^.aiFTrigActionTouchScreenNavPanel[5]:=0;
ptrConfigPage^.aiFTrigActionTouchScreenNavPanel[6]:=10460;
ptrConfigPage^.xMaskBtStart:=FALSE;
ptrConfigPage^.xMaskBtStop:=TRUE;

(* QVis page 470, Parameter Grind Axis *)
iIndexPage:=470;
iPageNumber:=iPageNumber+1;
T_Visu.T_PageIndex[iIndexPage].iIndexConfigPage:=iPageNumber;
ptrConfigPage:=ADR(T_Visu.T_ConfigPage[T_Visu.T_PageIndex[iIndexPage].iIndexConfigPage]);
ptrConfigPage^.sName:='Parameter Grind Axis';
ptrConfigPage^.wMaskBtPanelLeft:=16#1F;
ptrConfigPage^.wMaskBtPanelRight:=16#200;
ptrConfigPage^.wMaskFunctionPanel:=16#0;
(* Navigation panel restriction *)
ptrConfigPage^.wMaskTouchScreenNavPanel:=16#27;
(* Active machine movement mask *)
ptrConfigPage^.wMaskActiveMachineBtPanelLeft:=16#0;
ptrConfigPage^.wMaskActiveMachineBtPanelRight:=16#0;
ptrConfigPage^.wMaskActiveMachineFunctionPanel:=16#0;
ptrConfigPage^.wMaskActiveMachineNavPanel:=16#27;
(* Button edge action *)
ptrConfigPage^.aiRTrigActionPanelRight[1]:=0;
ptrConfigPage^.aiRTrigActionPanelRight[2]:=0;
ptrConfigPage^.aiRTrigActionPanelRight[3]:=0;
ptrConfigPage^.aiRTrigActionPanelRight[4]:=0;
ptrConfigPage^.aiRTrigActionPanelRight[5]:=1006;
ptrConfigPage^.aiFTrigActionPanelRight[1]:=0;
ptrConfigPage^.aiFTrigActionPanelRight[2]:=0;
ptrConfigPage^.aiFTrigActionPanelRight[3]:=0;
ptrConfigPage^.aiFTrigActionPanelRight[4]:=0;
ptrConfigPage^.aiFTrigActionPanelRight[5]:=0;
ptrConfigPage^.aiDelayActionPanelRight[1]:=0;
ptrConfigPage^.aiDelayActionPanelRight[2]:=0;
ptrConfigPage^.aiDelayActionPanelRight[3]:=0;
ptrConfigPage^.aiDelayActionPanelRight[4]:=0;
ptrConfigPage^.aiDelayActionPanelRight[5]:=0;
ptrConfigPage^.aiRTrigActionFunctionPanel[1]:=0;
ptrConfigPage^.aiRTrigActionFunctionPanel[2]:=0;
ptrConfigPage^.aiRTrigActionFunctionPanel[3]:=0;
ptrConfigPage^.aiRTrigActionFunctionPanel[4]:=0;
ptrConfigPage^.aiRTrigActionFunctionPanel[5]:=0;
ptrConfigPage^.aiRTrigActionFunctionPanel[6]:=0;
ptrConfigPage^.aiRTrigActionFunctionPanel[7]:=0;
ptrConfigPage^.aiRTrigActionFunctionPanel[8]:=0;
ptrConfigPage^.aiRTrigActionFunctionPanel[9]:=0;
ptrConfigPage^.aiRTrigActionFunctionPanel[10]:=0;
ptrConfigPage^.aiRTrigActionFunctionPanel[11]:=0;
ptrConfigPage^.aiRTrigActionFunctionPanel[12]:=0;
ptrConfigPage^.aiFTrigActionTouchScreenNavPanel[1]:=10410;
ptrConfigPage^.aiFTrigActionTouchScreenNavPanel[2]:=10420;
ptrConfigPage^.aiFTrigActionTouchScreenNavPanel[3]:=10430;
ptrConfigPage^.aiFTrigActionTouchScreenNavPanel[4]:=0;
ptrConfigPage^.aiFTrigActionTouchScreenNavPanel[5]:=0;
ptrConfigPage^.aiFTrigActionTouchScreenNavPanel[6]:=10460;
ptrConfigPage^.xMaskBtStart:=FALSE;
ptrConfigPage^.xMaskBtStop:=TRUE;
END_FUNCTION_BLOCK

(* POU PRG_VISU_LAYER5/FB_VISU/FB_COMPAREPROFILEPROCESSVALUE, ST *)
FUNCTION_BLOCK FB_COMPAREPROFILEPROCESSVALUE
VAR_INPUT
	T_Data_ProcessImageLoadData:ST_RETAIN_DATA_PROCESSIMAGE;	(* Novram parameter structure for the profile value *)
	T_Data_ProcessImageData:ST_RETAIN_DATA_PROCESSIMAGE;		(* Novram parametre structure for the process parameter *)
	xMicroRodActive: BOOL;											(* choice of the machine MicroWire or MicroRod *)
END_VAR
VAR_OUTPUT
	xProcessValueModified:BOOL;										(* TRUE=Profile parameter and process parameter are not the same, FALSE=both are same *)
END_VAR
VAR_IN_OUT
END_VAR
VAR
(* variable *)
	xFirstExecution:BOOL;
END_VAR
(****************************************************************************************************************************************************)
(***  This Functionblock check if the parameter of the loaded profile ar the same as the parameter of the process parameter   ***)
(****************************************************************************************************************************************************)
(* First execution *)
	IF NOT xFirstExecution THEN
		xProcessValueModified:=FALSE;
		(* confirm execution *)
		xFirstExecution:=TRUE;
	END_IF

(* compare value *)
	xProcessValueModified:=FALSE;

	(* value *)
	IF T_Data_ProcessImageLoadData.T_GeometryPara.arStartDiameter[1] <> T_Data_ProcessImageData.T_GeometryPara.arStartDiameter[1] THEN xProcessValueModified:=TRUE; RETURN; END_IF
	IF T_Data_ProcessImageLoadData.T_GeometryPara.arEndDiameter[1] <> T_Data_ProcessImageData.T_GeometryPara.arEndDiameter[1] THEN xProcessValueModified:=TRUE; RETURN; END_IF
	IF T_Data_ProcessImageLoadData.T_GeometryPara.arSectionLength[1] <> T_Data_ProcessImageData.T_GeometryPara.arSectionLength[1] THEN xProcessValueModified:=TRUE; RETURN; END_IF
	IF T_Data_ProcessImageLoadData.T_GeometryPara.arSectionPitch[1] <> T_Data_ProcessImageData.T_GeometryPara.arSectionPitch[1] THEN xProcessValueModified:=TRUE; RETURN; END_IF
	IF T_Data_ProcessImageLoadData.T_GeometryPara.axActiveSection[1] <> T_Data_ProcessImageData.T_GeometryPara.axActiveSection[1] THEN xProcessValueModified:=TRUE; RETURN; END_IF

	IF T_Data_ProcessImageLoadData.T_GeometryPara.arStartDiameter[2] <> T_Data_ProcessImageData.T_GeometryPara.arStartDiameter[2] THEN xProcessValueModified:=TRUE; RETURN; END_IF
	IF T_Data_ProcessImageLoadData.T_GeometryPara.arEndDiameter[2] <> T_Data_ProcessImageData.T_GeometryPara.arEndDiameter[2] THEN xProcessValueModified:=TRUE; RETURN; END_IF
	IF T_Data_ProcessImageLoadData.T_GeometryPara.arSectionLength[2] <> T_Data_ProcessImageData.T_GeometryPara.arSectionLength[2] THEN xProcessValueModified:=TRUE; RETURN; END_IF
	IF T_Data_ProcessImageLoadData.T_GeometryPara.arSectionPitch[2] <> T_Data_ProcessImageData.T_GeometryPara.arSectionPitch[2] THEN xProcessValueModified:=TRUE; RETURN; END_IF
	IF T_Data_ProcessImageLoadData.T_GeometryPara.axActiveSection[2] <> T_Data_ProcessImageData.T_GeometryPara.axActiveSection[2] THEN xProcessValueModified:=TRUE; RETURN; END_IF

	IF T_Data_ProcessImageLoadData.T_GeometryPara.arStartDiameter[3] <> T_Data_ProcessImageData.T_GeometryPara.arStartDiameter[3] THEN xProcessValueModified:=TRUE; RETURN; END_IF
	IF T_Data_ProcessImageLoadData.T_GeometryPara.arEndDiameter[3] <> T_Data_ProcessImageData.T_GeometryPara.arEndDiameter[3] THEN xProcessValueModified:=TRUE; RETURN; END_IF
	IF T_Data_ProcessImageLoadData.T_GeometryPara.arSectionLength[3] <> T_Data_ProcessImageData.T_GeometryPara.arSectionLength[3] THEN xProcessValueModified:=TRUE; RETURN; END_IF
	IF T_Data_ProcessImageLoadData.T_GeometryPara.arSectionPitch[3] <> T_Data_ProcessImageData.T_GeometryPara.arSectionPitch[3] THEN xProcessValueModified:=TRUE; RETURN; END_IF
	IF T_Data_ProcessImageLoadData.T_GeometryPara.axActiveSection[3] <> T_Data_ProcessImageData.T_GeometryPara.axActiveSection[3] THEN xProcessValueModified:=TRUE; RETURN; END_IF

	IF T_Data_ProcessImageLoadData.T_GeometryPara.arStartDiameter[4] <> T_Data_ProcessImageData.T_GeometryPara.arStartDiameter[4] THEN xProcessValueModified:=TRUE; RETURN; END_IF
	IF T_Data_ProcessImageLoadData.T_GeometryPara.arEndDiameter[4] <> T_Data_ProcessImageData.T_GeometryPara.arEndDiameter[4] THEN xProcessValueModified:=TRUE; RETURN; END_IF
	IF T_Data_ProcessImageLoadData.T_GeometryPara.arSectionLength[4] <> T_Data_ProcessImageData.T_GeometryPara.arSectionLength[4] THEN xProcessValueModified:=TRUE; RETURN; END_IF
	IF T_Data_ProcessImageLoadData.T_GeometryPara.arSectionPitch[4] <> T_Data_ProcessImageData.T_GeometryPara.arSectionPitch[4] THEN xProcessValueModified:=TRUE; RETURN; END_IF
	IF T_Data_ProcessImageLoadData.T_GeometryPara.axActiveSection[4] <> T_Data_ProcessImageData.T_GeometryPara.axActiveSection[4] THEN xProcessValueModified:=TRUE; RETURN; END_IF
(*09.12.2022: SOA *)
	IF T_Data_ProcessImageLoadData.T_GeometryPara.arStartDiameter[5] <> T_Data_ProcessImageData.T_GeometryPara.arStartDiameter[5] THEN xProcessValueModified:=TRUE; RETURN; END_IF
	IF T_Data_ProcessImageLoadData.T_GeometryPara.arEndDiameter[5] <> T_Data_ProcessImageData.T_GeometryPara.arEndDiameter[5] THEN xProcessValueModified:=TRUE; RETURN; END_IF
	IF T_Data_ProcessImageLoadData.T_GeometryPara.arSectionLength[5] <> T_Data_ProcessImageData.T_GeometryPara.arSectionLength[5] THEN xProcessValueModified:=TRUE; RETURN; END_IF
	IF T_Data_ProcessImageLoadData.T_GeometryPara.arSectionPitch[5] <> T_Data_ProcessImageData.T_GeometryPara.arSectionPitch[5] THEN xProcessValueModified:=TRUE; RETURN; END_IF
	IF T_Data_ProcessImageLoadData.T_GeometryPara.axActiveSection[5] <> T_Data_ProcessImageData.T_GeometryPara.axActiveSection[5] THEN xProcessValueModified:=TRUE; RETURN; END_IF

	IF T_Data_ProcessImageLoadData.T_GeometryPara.arStartDiameter[6] <> T_Data_ProcessImageData.T_GeometryPara.arStartDiameter[6] THEN xProcessValueModified:=TRUE; RETURN; END_IF
	IF T_Data_ProcessImageLoadData.T_GeometryPara.arEndDiameter[6] <> T_Data_ProcessImageData.T_GeometryPara.arEndDiameter[6] THEN xProcessValueModified:=TRUE; RETURN; END_IF
	IF T_Data_ProcessImageLoadData.T_GeometryPara.arSectionLength[6] <> T_Data_ProcessImageData.T_GeometryPara.arSectionLength[6] THEN xProcessValueModified:=TRUE; RETURN; END_IF
	IF T_Data_ProcessImageLoadData.T_GeometryPara.arSectionPitch[6] <> T_Data_ProcessImageData.T_GeometryPara.arSectionPitch[6] THEN xProcessValueModified:=TRUE; RETURN; END_IF
	IF T_Data_ProcessImageLoadData.T_GeometryPara.axActiveSection[6] <> T_Data_ProcessImageData.T_GeometryPara.axActiveSection[6] THEN xProcessValueModified:=TRUE; RETURN; END_IF
(*09.12.2022: SOA *)
	IF T_Data_ProcessImageLoadData.T_PrismPara.rPrismaDistanceD1 <> T_Data_ProcessImageData.T_PrismPara.rPrismaDistanceD1 THEN xProcessValueModified:=TRUE; RETURN; END_IF
	IF T_Data_ProcessImageLoadData.T_PrismPara.rPrismaDistanceD2 <> T_Data_ProcessImageData.T_PrismPara.rPrismaDistanceD2 THEN xProcessValueModified:=TRUE; RETURN; END_IF
	IF T_Data_ProcessImageLoadData.T_PrismPara.rPrismaAngleA <> T_Data_ProcessImageData.T_PrismPara.rPrismaAngleA THEN xProcessValueModified:=TRUE; RETURN; END_IF
	IF T_Data_ProcessImageLoadData.T_PrismPara.bStateInputPrisma <> T_Data_ProcessImageData.T_PrismPara.bStateInputPrisma THEN xProcessValueModified:=TRUE; RETURN; END_IF
	IF T_Data_ProcessImageLoadData.T_PrismPara.rToolDiameterMin <> T_Data_ProcessImageData.T_PrismPara.rToolDiameterMin THEN xProcessValueModified:=TRUE; RETURN; END_IF
	IF T_Data_ProcessImageLoadData.T_PrismPara.rToolDiameterMax <> T_Data_ProcessImageData.T_PrismPara.rToolDiameterMax THEN xProcessValueModified:=TRUE; RETURN; END_IF
	IF T_Data_ProcessImageLoadData.T_PrismPara.rPrismaFactor <> T_Data_ProcessImageData.T_PrismPara.rPrismaFactor THEN xProcessValueModified:=TRUE; RETURN; END_IF

	IF T_Data_ProcessImageLoadData.T_ProcessPara.rOffsetBeforeToolDiaGrindFeedProcess <> T_Data_ProcessImageData.T_ProcessPara.rOffsetBeforeToolDiaGrindFeedProcess THEN xProcessValueModified:=TRUE; RETURN; END_IF
	IF T_Data_ProcessImageLoadData.T_ProcessPara.rSecurityPosGrindFeedProcess <> T_Data_ProcessImageData.T_ProcessPara.rSecurityPosGrindFeedProcess THEN xProcessValueModified:=TRUE; RETURN; END_IF
	IF T_Data_ProcessImageLoadData.T_ProcessPara.rSpeedBackwardGrindFeed <> T_Data_ProcessImageData.T_ProcessPara.rSpeedBackwardGrindFeed THEN xProcessValueModified:=TRUE; RETURN; END_IF
	IF T_Data_ProcessImageLoadData.T_ProcessPara.rSpeedForwardFastGrindFeed <> T_Data_ProcessImageData.T_ProcessPara.rSpeedForwardFastGrindFeed THEN xProcessValueModified:=TRUE; RETURN; END_IF
	IF T_Data_ProcessImageLoadData.T_ProcessPara.rSpeedForwardSlowGrindFeed <> T_Data_ProcessImageData.T_ProcessPara.rSpeedForwardSlowGrindFeed THEN xProcessValueModified:=TRUE; RETURN; END_IF
	IF xMicroRodActive THEN
		IF T_Data_ProcessImageLoadData.T_ProcessPara.rSpeedStartPosToolFeedProcess <> T_Data_ProcessImageData.T_ProcessPara.rSpeedStartPosToolFeedProcess THEN xProcessValueModified:=TRUE; RETURN; END_IF
		IF T_Data_ProcessImageLoadData.T_ProcessPara.rStartPosToolFeedAuto <> T_Data_ProcessImageData.T_ProcessPara.rStartPosToolFeedAuto THEN xProcessValueModified:=TRUE; RETURN; END_IF
	END_IF;
	IF T_Data_ProcessImageLoadData.T_ProcessPara.rToolDiameterProcess <> T_Data_ProcessImageData.T_ProcessPara.rToolDiameterProcess THEN xProcessValueModified:=TRUE; RETURN; END_IF
	IF T_Data_ProcessImageLoadData.T_ProcessPara.rToolTensionProcess <> T_Data_ProcessImageData.T_ProcessPara.rToolTensionProcess THEN xProcessValueModified:=TRUE; RETURN; END_IF

	IF T_Data_ProcessImageLoadData.T_AutoGeometryPara.iCycleGeometry <> T_Data_ProcessImageData.T_AutoGeometryPara.iCycleGeometry THEN xProcessValueModified:=TRUE; RETURN; END_IF
	IF xMicroRodActive THEN
		IF T_Data_ProcessImageLoadData.T_AutoGeometryPara.rPlungeCycleGrindFeedGeometry <> T_Data_ProcessImageData.T_AutoGeometryPara.rPlungeCycleGrindFeedGeometry THEN xProcessValueModified:=TRUE; RETURN; END_IF
	END_IF;
	IF T_Data_ProcessImageLoadData.T_AutoGeometryPara.rDisplaceLengthToolFeedGeometry <> T_Data_ProcessImageData.T_AutoGeometryPara.rDisplaceLengthToolFeedGeometry THEN xProcessValueModified:=TRUE; RETURN; END_IF
	IF T_Data_ProcessImageLoadData.T_AutoGeometryPara.rDisplaceSpeedGrindFeedGeometry <> T_Data_ProcessImageData.T_AutoGeometryPara.rDisplaceSpeedGrindFeedGeometry THEN xProcessValueModified:=TRUE; RETURN; END_IF
	IF T_Data_ProcessImageLoadData.T_AutoGeometryPara.rPlungeLengthToolFeedGeometry <> T_Data_ProcessImageData.T_AutoGeometryPara.rPlungeLengthToolFeedGeometry THEN xProcessValueModified:=TRUE; RETURN; END_IF
	IF T_Data_ProcessImageLoadData.T_AutoGeometryPara.rPlungeSpeedGrindFeedGeometry <> T_Data_ProcessImageData.T_AutoGeometryPara.rPlungeSpeedGrindFeedGeometry THEN xProcessValueModified:=TRUE; RETURN; END_IF
	IF T_Data_ProcessImageLoadData.T_AutoGeometryPara.rSpeedToolRotationGeometry <> T_Data_ProcessImageData.T_AutoGeometryPara.rSpeedToolRotationGeometry THEN xProcessValueModified:=TRUE; RETURN; END_IF
	IF T_Data_ProcessImageLoadData.T_AutoGeometryPara.xDisplaceActivationGeometry <> T_Data_ProcessImageData.T_AutoGeometryPara.xDisplaceActivationGeometry THEN xProcessValueModified:=TRUE; RETURN; END_IF
	IF T_Data_ProcessImageLoadData.T_AutoGeometryPara.xPlungeActivationGeometry <> T_Data_ProcessImageData.T_AutoGeometryPara.xPlungeActivationGeometry THEN xProcessValueModified:=TRUE; RETURN; END_IF

	IF T_Data_ProcessImageLoadData.T_AutoGroovePara.rDisplaceLengthToolFeedGroove <> T_Data_ProcessImageData.T_AutoGroovePara.rDisplaceLengthToolFeedGroove THEN xProcessValueModified:=TRUE; RETURN; END_IF
	IF T_Data_ProcessImageLoadData.T_AutoGroovePara.rDisplaceSpeedGrindFeedGroove <> T_Data_ProcessImageData.T_AutoGroovePara.rDisplaceSpeedGrindFeedGroove THEN xProcessValueModified:=TRUE; RETURN; END_IF
	IF T_Data_ProcessImageLoadData.T_AutoGroovePara.rPitchGroove <> T_Data_ProcessImageData.T_AutoGroovePara.rPitchGroove THEN xProcessValueModified:=TRUE; RETURN; END_IF
	IF T_Data_ProcessImageLoadData.T_AutoGroovePara.rPlungeLengthToolFeedGroove <> T_Data_ProcessImageData.T_AutoGroovePara.rPlungeLengthToolFeedGroove THEN xProcessValueModified:=TRUE; RETURN; END_IF
	IF T_Data_ProcessImageLoadData.T_AutoGroovePara.rPlungeSpeedGrindFeedGroove <> T_Data_ProcessImageData.T_AutoGroovePara.rPlungeSpeedGrindFeedGroove THEN xProcessValueModified:=TRUE; RETURN; END_IF
	IF T_Data_ProcessImageLoadData.T_AutoGroovePara.rSpeedToolRotationGroove <> T_Data_ProcessImageData.T_AutoGroovePara.rSpeedToolRotationGroove THEN xProcessValueModified:=TRUE; RETURN; END_IF
	IF T_Data_ProcessImageLoadData.T_AutoGroovePara.xDisplaceActivationGroove <> T_Data_ProcessImageData.T_AutoGroovePara.xDisplaceActivationGroove THEN xProcessValueModified:=TRUE; RETURN; END_IF
	IF T_Data_ProcessImageLoadData.T_AutoGroovePara.xPlungeActivationGroove <> T_Data_ProcessImageData.T_AutoGroovePara.xPlungeActivationGroove THEN xProcessValueModified:=TRUE; RETURN; END_IF
	IF T_Data_ProcessImageLoadData.T_AutoGroovePara.xBlockGrindFeeder <> T_Data_ProcessImageData.T_AutoGroovePara.xBlockGrindFeeder THEN xProcessValueModified:=TRUE; RETURN; END_IF
	IF T_Data_ProcessImageLoadData.T_AutoGroovePara.iNumberOfGrooves <> T_Data_ProcessImageData.T_AutoGroovePara.iNumberOfGrooves THEN xProcessValueModified:=TRUE; RETURN; END_IF

	IF T_Data_ProcessImageLoadData.T_CalibrationPara.rDisplaceLengthToolFeedCalib <> T_Data_ProcessImageData.T_CalibrationPara.rDisplaceLengthToolFeedCalib THEN xProcessValueModified:=TRUE; RETURN; END_IF
	IF T_Data_ProcessImageLoadData.T_CalibrationPara.rDisplaceSpeedGrindFeedCalib <> T_Data_ProcessImageData.T_CalibrationPara.rDisplaceSpeedGrindFeedCalib THEN xProcessValueModified:=TRUE; RETURN; END_IF
	IF NOT(xMicroRodActive) THEN
		IF T_Data_ProcessImageLoadData.T_CalibrationPara.rMeasureOffsetToolFeedCalib <> T_Data_ProcessImageData.T_CalibrationPara.rMeasureOffsetToolFeedCalib THEN xProcessValueModified:=TRUE; RETURN; END_IF
	END_IF;
	IF xMicroRodActive THEN
		IF T_Data_ProcessImageLoadData.T_CalibrationPara.rMeasurePosToolFeedCalib <> T_Data_ProcessImageData.T_CalibrationPara.rMeasurePosToolFeedCalib THEN xProcessValueModified:=TRUE; RETURN; END_IF
		IF T_Data_ProcessImageLoadData.T_CalibrationPara.rStartPosToolFeedCalib <> T_Data_ProcessImageData.T_CalibrationPara.rStartPosToolFeedCalib THEN xProcessValueModified:=TRUE; RETURN; END_IF
	END_IF;
	IF T_Data_ProcessImageLoadData.T_CalibrationPara.rPitchCalib <> T_Data_ProcessImageData.T_CalibrationPara.rPitchCalib THEN xProcessValueModified:=TRUE; RETURN; END_IF
	IF T_Data_ProcessImageLoadData.T_CalibrationPara.rPlungeLengthGrindFeedCalib <> T_Data_ProcessImageData.T_CalibrationPara.rPlungeLengthGrindFeedCalib THEN xProcessValueModified:=TRUE; RETURN; END_IF
	IF T_Data_ProcessImageLoadData.T_CalibrationPara.rPlungeLengthToolFeedCalib <> T_Data_ProcessImageData.T_CalibrationPara.rPlungeLengthToolFeedCalib THEN xProcessValueModified:=TRUE; RETURN; END_IF
	IF T_Data_ProcessImageLoadData.T_CalibrationPara.rPlungeSpeedGrindFeedCalib <> T_Data_ProcessImageData.T_CalibrationPara.rPlungeSpeedGrindFeedCalib THEN xProcessValueModified:=TRUE; RETURN; END_IF
	IF T_Data_ProcessImageLoadData.T_CalibrationPara.rSpeedToolRotationCalib <> T_Data_ProcessImageData.T_CalibrationPara.rSpeedToolRotationCalib THEN xProcessValueModified:=TRUE; RETURN; END_IF
	IF T_Data_ProcessImageLoadData.T_CalibrationPara.rToolLengthCylinderPartCalib <> T_Data_ProcessImageData.T_CalibrationPara.rToolLengthCylinderPartCalib THEN xProcessValueModified:=TRUE; RETURN; END_IF
	IF T_Data_ProcessImageLoadData.T_CalibrationPara.xDisplaceActivationCalib <> T_Data_ProcessImageData.T_CalibrationPara.xDisplaceActivationCalib THEN xProcessValueModified:=TRUE; RETURN; END_IF
	IF T_Data_ProcessImageLoadData.T_CalibrationPara.xPlungeActivationCalib <> T_Data_ProcessImageData.T_CalibrationPara.xPlungeActivationCalib THEN xProcessValueModified:=TRUE; RETURN; END_IF
END_FUNCTION_BLOCK

(* POU PRG_VISU_LAYER5/FB_VISU/FB_CALC_TORQUE, ST *)
FUNCTION_BLOCK FB_CALC_TORQUE
VAR_INPUT
	xStart:BOOL;				(* start the calculation of the mean value of the torque *)
	uiActualTorque:UINT;		(* actual current value *)
	uiZeroTorque:UINT;		(* set value of the current value for scale the range *)
	iStepCalc:INT;			(* number of mean value *)
END_VAR
VAR_OUTPUT
	uiCalcTorque:UINT;		(* calculated torque value in % of the maximal torque of the motor *)
END_VAR
VAR
	auiSaveTorque: ARRAY [1..200] OF UINT;
	auiTmpSaveTorque: ARRAY [1..200] OF UINT;
	auiDeleteTorque: ARRAY [1..200] OF UINT;
	uiSumTorque: UINT;
	ii: INT;
	xInit: BOOL;
	uiTmpZeroTorque:UINT;
	rMaxMotorCurrent: REAL;
	rMaxMotorTorque: REAL;
END_VAR
(****************************************************************************************************************************************************)
(***********             This Functionblock calc the torque of the ToolRotation with set and reset torque function                         ************)
(****************************************************************************************************************************************************)
uiCalcTorque:=0;
IF NOT(xStart) AND xInit THEN
	xInit:=FALSE;
	auiSaveTorque:=auiDeleteTorque;
	auiTmpSaveTorque:=auiDeleteTorque;
	uiTmpZeroTorque:=uiZeroTorque;
END_IF;
IF xStart THEN
	xInit:=TRUE;
	uiSumTorque:=0;
	IF (uiZeroTorque <> uiTmpZeroTorque) THEN
		auiSaveTorque:=auiDeleteTorque;
		auiTmpSaveTorque:=auiDeleteTorque;
		uiTmpZeroTorque:=uiZeroTorque;
	END_IF;
	IF (iStepCalc > 0) AND (iStepCalc <= 200) THEN
		FOR ii:=1 TO (iStepCalc - 1)  DO
			auiTmpSaveTorque[ii+1]:=auiSaveTorque[ii];
			uiSumTorque:=uiSumTorque + auiSaveTorque[ii];
		END_FOR;
		auiSaveTorque:=auiTmpSaveTorque;
		IF (uiTmpZeroTorque <= uiActualTorque) THEN
			auiSaveTorque[1]:=uiActualTorque - uiTmpZeroTorque;
		ELSE
			auiSaveTorque[1]:=0;
		END_IF;
		uiSumTorque:=uiSumTorque + auiSaveTorque[1];
		uiSumTorque:=uiSumTorque/iStepCalc;
		rMaxMotorCurrent:=6.0;	(* EcoStep Motor 23S21  *)
		rMaxMotorTorque:=(rMaxMotorCurrent * 0.16) * 1000.0;	(* 0.16 = 0.16Nm/A -->1000.0= Umwandlung in mNm *)
		uiCalcTorque:=REAL_TO_UINT((UINT_TO_REAL(uiSumTorque) / (REAL_TO_UINT(rMaxMotorTorque) - uiTmpZeroTorque)) * 100.0);	(* Ausgabe in % des Max Stromes *)
		IF (uiCalcTorque >= 100) THEN
			uiCalcTorque:=100;
		END_IF;
	END_IF;
END_IF;
END_FUNCTION_BLOCK

(* POU PRG_VISU_LAYER5/FB_VISU/FBQVIS_ERROR_LIST, ST *)
FUNCTION_BLOCK FBQVIS_ERROR_LIST
VAR_INPUT
	T_ErrorList:ST_ERROR_LIST;					(* Static define Error List *)
	T_ErrorNrList:ST_RETAIN_ERROR_DATA;		(* Daten welche im NOVram abgelegt sind *)
END_VAR
VAR_IN_OUT
	T_MsgErrorEnglish:ST_EXCHG_MESSAGE_ERROR;	(* Daten die auf der Visu in der Errorliste visualisiert werden *)
	T_MsgErrorDeutsch:ST_EXCHG_MESSAGE_ERROR;	(* Daten die auf der Visu in der Errorliste visualisiert werden *)
	T_MsgErrorFrancais:ST_EXCHG_MESSAGE_ERROR;	(* Daten die auf der Visu in der Errorliste visualisiert werden *)
END_VAR
VAR_OUTPUT
END_VAR
VAR
	FBErrorMessage:FB_ErrorMessage;
	ii:INT;
	diErrorNr: DINT;
	sErrorTimeStamp: STRING(12);
END_VAR
(****************************************************************************************************************************************************)
(***********                              This Functionblock fills the errorlist with the errormesse and the timestamp                                  ************)
(****************************************************************************************************************************************************)
	FOR ii:=1 TO 20 DO
		diErrorNr:=T_ErrorNrList.adiErrorListMachine[ii];
		sErrorTimeStamp:=T_ErrorNrList.asErrorTimeStampMachine[ii];
		sErrorTimeStamp:=CONCAT(sErrorTimeStamp,'--');
		IF (diErrorNr <> 0) THEN
			FBErrorMessage(	diErrorNr:=diErrorNr ,
							T_ErrorList:=T_ErrorList);
			T_MsgErrorEnglish.asMsgErrorList[ii]:=CONCAT(sErrorTimeStamp,FBErrorMessage.sErrorTextEnglish);
			T_MsgErrorDeutsch.asMsgErrorList[ii]:=CONCAT(sErrorTimeStamp,FBErrorMessage.sErrorTextDeutsch);
			T_MsgErrorFrancais.asMsgErrorList[ii]:=CONCAT(sErrorTimeStamp,FBErrorMessage.sErrorTextFrancais);
		ELSE
			T_MsgErrorEnglish.asMsgErrorList[ii]:='                                                                    ';
			T_MsgErrorDeutsch.asMsgErrorList[ii]:='                                                                    ';
			T_MsgErrorFrancais.asMsgErrorList[ii]:='                                                                    ';
		END_IF;
	END_FOR;
END_FUNCTION_BLOCK

(* POU PRG_VISU_LAYER5/FB_VISU/FB_SETERRORLIST, ST *)
FUNCTION_BLOCK FB_SETERRORLIST
VAR_INPUT
	TControlStation : ST_CONTROL;					(* Control structur of the data station structure *)
	TProcess : ST_PROCESS;						(* data structure of the processlevel *)
END_VAR
VAR_IN_OUT
	xParameterSaved:BOOL;						(* state, if the changed errorlist was saved *)
	T_ErrorNrList:ST_RETAIN_ERROR_DATA;		(* Daten welche im NOVram abgelegt sind *)
	xSetForceError:BOOL;							(* manual input of an error into the error list *)
	diSetForceErrorNr:DINT;						(* manual input of an error number into the error list *)
END_VAR
VAR_OUTPUT
	xSaveParameter:BOOL;						(* save the maked or updated error list into the Novram *)
END_VAR
VAR
	xTmpStation: BOOL;
	xTmpProcess: BOOL;
	iTmpStationNr:INT;
	xBlockProcessProc: BOOL;
	xBlockStationProc: BOOL;
	adiTmpErrorList: ARRAY [1..20] OF DINT;
	asTmpErrorList: ARRAY [1..20] OF STRING(12);
	ii:INT;
	xDataChanged: BOOL;
	xQuitError: BOOL;
	TimerCheckQuitError:TON;
	FBNT_GetTime:NT_GetTime;
	xUpdateProcTimeStamp:BOOL;
	xInitGetTime: BOOL;
END_VAR
(****************************************************************************************************************************************************)
(***********                       This Functionblock manage the machine error, for make and update the errorlist                             ************)
(****************************************************************************************************************************************************)
xTmpStation:=TControlStation.xError AND TControlStation.xActiveStation;
xTmpProcess:=TProcess.xError AND TProcess.xRdy;

IF NOT(xDataChanged) THEN
	IF NOT(TProcess.xEnd) AND TProcess.xError AND NOT(xBlockProcessProc) AND NOT(xBlockStationProc) AND NOT(xSetForceError) THEN
		xBlockProcessProc:=TRUE;
		iTmpStationNr:=0;
	END_IF;
	IF TProcess.xEnd AND xTmpStation AND NOT(xBlockStationProc) AND NOT(xBlockProcessProc) AND NOT(xSetForceError) THEN
		xBlockStationProc:=TRUE;
		iTmpStationNr:=1;
	END_IF;
	IF xBlockProcessProc AND NOT(xQuitError) THEN
		adiTmpErrorList:=T_ErrorNrList.adiErrorListMachine;
		T_ErrorNrList.adiErrorListMachine[1]:=TProcess.diErrorNr;
		FOR ii:=2 TO 20 DO
			T_ErrorNrList.adiErrorListMachine[ii]:=adiTmpErrorList[ii-1];
		END_FOR;
		xUpdateProcTimeStamp:=TRUE;
	END_IF;
	
	IF xBlockStationProc AND NOT(xQuitError) THEN
		adiTmpErrorList:=T_ErrorNrList.adiErrorListMachine;
		T_ErrorNrList.adiErrorListMachine[1]:=TControlStation.diErrorNr;
		FOR ii:=2 TO 20 DO
			T_ErrorNrList.adiErrorListMachine[ii]:=adiTmpErrorList[ii-1];
		END_FOR;
		xUpdateProcTimeStamp:=TRUE;
	END_IF;
	
	IF xSetForceError AND NOT(xQuitError) AND NOT(xBlockStationProc) AND NOT(xBlockProcessProc) THEN
		adiTmpErrorList:=T_ErrorNrList.adiErrorListMachine;
		T_ErrorNrList.adiErrorListMachine[1]:=diSetForceErrorNr;
		FOR ii:=2 TO 20 DO
			T_ErrorNrList.adiErrorListMachine[ii]:=adiTmpErrorList[ii-1];
		END_FOR;
		xUpdateProcTimeStamp:=TRUE;
		xSetForceError:=FALSE;
	ELSE
		xSetForceError:=FALSE;
	END_IF;

	IF xUpdateProcTimeStamp THEN
		IF NOT(xInitGetTime) THEN
			xInitGetTime:=TRUE;
			FBNT_GetTime(	NETID:= '',
							START:=FALSE );
		END_IF;
		FBNT_GetTime(	NETID:= '',
						START:= TRUE,
						TMOUT:= T#2s);
		IF NOT(FBNT_GetTime.BUSY) OR FBNT_GetTime.ERR THEN
			IF xUpdateProcTimeStamp THEN
				asTmpErrorList:=T_ErrorNrList.asErrorTimeStampMachine;
				IF NOT(FBNT_GetTime.ERR) THEN
					T_ErrorNrList.asErrorTimeStampMachine[1]:=Fct_ConvertDateToString(2,FBNT_GetTime.TIMESTR);
				ELSE
					T_ErrorNrList.asErrorTimeStampMachine[1]:='00.00 00:00';	(* Fehler beim lesen der Systemzeit, daher wird ein default-Wert gesetzt *)
				END_IF;
				FOR ii:=2 TO 20 DO
					T_ErrorNrList.asErrorTimeStampMachine[ii]:=asTmpErrorList[ii-1];
				END_FOR;
			END_IF;
			xInitGetTime:=FALSE;
			xUpdateProcTimeStamp:=FALSE;
			xDataChanged:=TRUE;
		END_IF;
	END_IF;
END_IF;

IF xBlockProcessProc OR xBlockStationProc THEN
	xQuitError:=TRUE;
	IF TControlStation.xQuitError OR TProcess.xQuitError THEN
		xBlockProcessProc:=xBlockStationProc:=xSetForceError:=xQuitError:=FALSE;
	END_IF;
	IF NOT(xTmpStation) AND NOT(xTmpProcess) THEN
		TimerCheckQuitError(IN:=TRUE,PT:=T#1s);
		IF TimerCheckQuitError.Q THEN
			TimerCheckQuitError(IN:=FALSE);
			xBlockProcessProc:=xBlockStationProc:=xSetForceError:=xQuitError:=FALSE;
		END_IF;
	ELSE
		TimerCheckQuitError(IN:=FALSE);
	END_IF;
ELSE
	xQuitError:=FALSE;
END_IF;

IF xDataChanged THEN
	xSaveParameter:=TRUE;
	IF xParameterSaved THEN
		xParameterSaved:=xDataChanged:=xSaveParameter:=FALSE;
	END_IF;
END_IF;
END_FUNCTION_BLOCK

(* POU PRG_PROCESS_LAYER4/FB_PROCESS/Fct_ConvertDateToString, ST *)
FUNCTION Fct_ConvertDateToString : STRING
VAR_INPUT
		iFormat:INT;	(* 0=Langes Date-Time Format; 1=Kurzes Date-Time Format; 2=Sehr Kurzes Date-Time Format *)
					(* 0='28.March 2007  08:47:01' *)
					(* 1='28.03.07 08:47' *)
					(* 2='28.03 08:47' *)
		TProcTimeStart:TIMESTRUCT;
END_VAR
VAR
	sTmpData:STRING(255);
	sTmpData1:STRING(255);
	wYear: WORD;
END_VAR
(****************************************************************************************************************************************************)
(***********                                This Functionblock formate a Date and Time String DD:MM HH:MM:SS                                     ************)
(****************************************************************************************************************************************************)
sTmpData:=sTmpData1:='';
IF (iFormat < 0) OR (iFormat > 2) THEN
	sTmpData1:='Wrong Date';
	Fct_ConvertDateToString:=sTmpData1;
	RETURN;
END_IF;
IF (TProcTimeStart.wDay <> 0) THEN
	IF (TProcTimeStart.wDay >= 0) AND (TProcTimeStart.wDay <= 9) THEN
		sTmpData1:=MUX(TProcTimeStart.wDay,'00','01','02','03','04','05','06','07','08','09');
		sTmpData:=CONCAT(sTmpData,sTmpData1);
	ELSE
		sTmpData:=CONCAT(sTmpData,WORD_TO_STRING(TProcTimeStart.wDay));
	END_IF;
	sTmpData:=CONCAT(sTmpData,'.');
ELSE
	sTmpData1:='Wrong Date';
	Fct_ConvertDateToString:=sTmpData1;
	RETURN;
END_IF;
IF (TProcTimeStart.wMonth <> 0) THEN
	IF (iFormat = 0) THEN
		sTmpData1:=MUX(TProcTimeStart.wMonth-1,'January','February','March','April','May','June','July','August','September','October','November','December');
	END_IF;
	IF (iFormat = 1) OR (iFormat = 2) THEN
		sTmpData1:=MUX(TProcTimeStart.wMonth-1,'01','02','03','04','05','06','07','08','09','10','11','12');
	END_IF;
ELSE
	sTmpData1:='Wrong Date';
	Fct_ConvertDateToString:=sTmpData1;
	RETURN;
END_IF;
sTmpData:=CONCAT(sTmpData,sTmpData1);
IF (iFormat = 0) THEN
	sTmpData:=CONCAT(sTmpData,' ');
END_IF;
IF (iFormat = 1) THEN
	sTmpData:=CONCAT(sTmpData,'.');
END_IF;
IF (iFormat = 2) THEN
	sTmpData:=CONCAT(sTmpData,' ');
END_IF;
IF (iFormat = 0) OR (iFormat = 1) THEN
	IF (TProcTimeStart.wYear <> 0) THEN
		IF (iFormat = 0) THEN
			sTmpData:=CONCAT(sTmpData,WORD_TO_STRING(TProcTimeStart.wYear));
			sTmpData:=CONCAT(sTmpData,'  ');
		END_IF;
		IF (iFormat = 1) THEN
			IF (TProcTimeStart.wYear >= 1000) AND (TProcTimeStart.wYear < 2000) THEN
				wYear:=TProcTimeStart.wYear - 1000;
			END_IF;
			IF (TProcTimeStart.wYear >= 2000) AND (TProcTimeStart.wYear < 3000) THEN
				wYear:=TProcTimeStart.wYear - 2000;
			END_IF;
			IF (wYear >= 0) AND (wYear < 10) THEN
				sTmpData1:=MUX(wYear,'00','01','02','03','04','05','06','07','08','09');
				sTmpData:=CONCAT(sTmpData,sTmpData1);
			ELSE
				sTmpData:=CONCAT(sTmpData,WORD_TO_STRING(wYear));
			END_IF;
			sTmpData:=CONCAT(sTmpData,' ');
		END_IF;
	ELSE
		sTmpData1:='Wrong Date';
		Fct_ConvertDateToString:=sTmpData1;
		RETURN;
	END_IF;
END_IF;
IF (TProcTimeStart.wHour >= 0) AND (TProcTimeStart.wHour <= 9) THEN
	sTmpData1:=MUX(TProcTimeStart.wHour,'00','01','02','03','04','05','06','07','08','09');
	sTmpData:=CONCAT(sTmpData,sTmpData1);
ELSE
	sTmpData:=CONCAT(sTmpData,WORD_TO_STRING(TProcTimeStart.wHour));
END_IF;
sTmpData:=CONCAT(sTmpData,':');
IF (TProcTimeStart.wMinute >= 0) AND (TProcTimeStart.wMinute <= 9) THEN
	sTmpData1:=MUX(TProcTimeStart.wMinute,'00','01','02','03','04','05','06','07','08','09');
	sTmpData:=CONCAT(sTmpData,sTmpData1);
ELSE
	sTmpData:=CONCAT(sTmpData,WORD_TO_STRING(TProcTimeStart.wMinute));
END_IF;
IF (iFormat = 0) THEN
	sTmpData:=CONCAT(sTmpData,':');
	IF (TProcTimeStart.wSecond >= 0) AND (TProcTimeStart.wSecond <= 9) THEN
		sTmpData1:=MUX(TProcTimeStart.wSecond,'00','01','02','03','04','05','06','07','08','09');
		sTmpData:=CONCAT(sTmpData,sTmpData1);
	ELSE
		sTmpData:=CONCAT(sTmpData,WORD_TO_STRING(TProcTimeStart.wSecond));
	END_IF;
END_IF;
Fct_ConvertDateToString:=sTmpData;
END_FUNCTION

(* POU PRG_VISU_LAYER5/FB_VISU/FBQVIS_CLEARERROR, ST *)
FUNCTION_BLOCK FBQVIS_CLEARERROR
VAR_INPUT
	xExecute:BOOL;				(* quit the error *)
	iError:INT;					(* occured error number *)
END_VAR
VAR_IN_OUT
	T_Message:ST_EXCHG_MESSAGE;		(* data structure for the message handling *)
	T_Station:ST_STATION;				(* data structure for the stationlevel *)
	T_Process : ST_PROCESS;			(* data structure for the processlevel *)
	T_NovRAM:ST_NOVRAM;				(* data structure for the Novram *)
	T_Profile:ST_PROFILE;				(* data structure for the profile management *)
	T_HDD:ST_HDD;						(* data structure for the file management *)
END_VAR
VAR_OUTPUT
	xDone:BOOL;
	xNotReady:BOOL;
	xErr:BOOL;
	udiErrorID:UDINT;
END_VAR
VAR
(* Trigger *)
	RisingEdgeExecute:R_TRIG;
(* Pointer *)
	ptrActivStation:POINTER TO ST_STATION;
(* Variable *)
	xClearError_Done:BOOL;
	xClearError_Err:BOOL;
	xClearError_NotReady:BOOL;
	xStepClearDone:BOOL;
	udiClearError_ErrorID:UDINT;
	iStepClearErrorStation:INT;
	iStepClearErrorMachine:INT;
	iStepClearStandardError: INT;
	xClearProcess:BOOL;
	xClearStation:BOOL;
	xClearStandardError:BOOL;
	xClearConifgErrStation: BOOL;
	xTmp: BOOL;
	xClearAxis: BOOL;
	iStepClearErrorAxis: INT;
	xTmp1: BOOL;
	xActiveMicroRod: BOOL;
	iTryAgain: INT;
END_VAR
(****************************************************************************************************************************************************)
(***********              This Functionblock manage an occured machine error so that the right component are quittet              ************)
(****************************************************************************************************************************************************)
	IF (T_NovRAM.T_Data.T_Standard.T_MachineConfig.iConfigMachineType = 2) THEN
		xActiveMicroRod:=TRUE;
	ELSE
		xActiveMicroRod:=FALSE;
	END_IF;

	RisingEdgeExecute(CLK:=xExecute);
	IF RisingEdgeExecute.Q THEN
	(* Init. variable by start clear error *)
		(* ...output *)
		xDone:=FALSE;
		xNotReady:=FALSE;
		xErr:=FALSE;
		udiErrorID:=16#0;
		(* ...variable *)
		xClearError_Done:=FALSE;
		xClearError_Err:=FALSE;
		xClearError_NotReady:=FALSE;
		xStepClearDone:=FALSE;
		iStepClearErrorStation:=1;
		iStepClearErrorMachine:=1;
		iStepClearStandardError:=1;
		iStepClearErrorAxis:=1;
		(* determin clear action *)
		xClearProcess:=xClearStation:=xClearAxis:=xClearStandardError:=FALSE;
		xClearConifgErrStation:=FALSE;
		IF T_Process.xError THEN
			xClearProcess:=TRUE;
		ELSE
			IF T_Station.TControl.xError AND NOT(T_Station.TControl.xEnd) THEN ptrActivStation:=ADR(T_Station); xClearStation:=TRUE; END_IF
			xTmp:=	(T_Station.THardware.TAxisToolLeft.T_CtrleSingle.xErr OR
					(T_Station.THardware.TAxisToolCenter.T_CtrleSingle.xErr AND xActiveMicroRod) OR
					T_Station.THardware.TAxisToolRight.T_CtrleSingle.xErr OR
					T_Station.THardware.TAxisToolFeeder.T_CtrleSingle.xErr OR
					T_Station.THardware.TAxisGrindFeeder.T_CtrleSingle.xErr) AND
					NOT(xClearStation);
			IF xTmp THEN
				xClearAxis:=TRUE;
			END_IF;
			IF T_Station.TControl.xError AND T_Station.TControl.xEnd AND NOT(xClearAxis) THEN
				xClearConifgErrStation:=TRUE;
			END_IF
		END_IF
		IF NOT xClearProcess AND NOT xClearStation AND NOT xClearConifgErrStation AND NOT xClearAxis THEN xClearStandardError:=TRUE; END_IF
		(* Exit FB *)
		RETURN;
	END_IF

	IF xClearProcess THEN
	(* Reset Error machine *)
		CASE iStepClearErrorMachine OF
		(* check station *)
		1:	IF T_Process.xError THEN iStepClearErrorMachine:=10; ELSE iStepClearErrorMachine:=90; END_IF
		(* activ clear error *)
		10:	T_Process.xQuitError:=TRUE;
			(* next step *)
			iStepClearErrorMachine:=20;
			xStepClearDone:=FALSE;
		(* waiting end clearing error *)
		20:	IF NOT T_Process.xQuitError THEN
				iStepClearErrorMachine:=90;
				xStepClearDone:=FALSE;
			END_IF
			IF T_Process.xError THEN iStepClearErrorMachine:=90; END_IF
		(* Clear error station done *)
		90:	xClearError_Done:=TRUE;
		(* Error *)
		99:	xClearError_Err:=TRUE;
		END_CASE
	END_IF

	IF xClearStation THEN
	(* Reset Error station *)
		CASE iStepClearErrorStation OF
		(* check station *)
		1:	IF ptrActivStation^.TControl.xError THEN iStepClearErrorStation:=10;
			ELSE IStepClearErrorStation:=90; END_IF
		(* activ clear error *)
		10:	ptrActivStation^.TControl.xQuitError:=TRUE;
			(* next step *)
			iStepClearErrorStation:=20;
			xStepClearDone:=FALSE;
		(* waiting end clearing error *)
		20:	IF NOT(xStepClearDone) THEN
			(* release action *)
				ptrActivStation^.TControl.xQuitError:=FALSE;
				xStepClearDone:=TRUE;
			ELSE
				IF ptrActivStation^.TControl.xEnd THEN
				(* confirm clear error, next step *)
					iStepClearErrorStation:=90;
					xStepClearDone:=FALSE;
				END_IF
				IF ptrActivStation^.TControl.xError THEN iStepClearErrorStation:=99; END_IF
			END_IF
		(* Clear error station done *)
		90:	xClearError_Done:=TRUE;
		(* Error *)
		99:	xClearError_Done:=TRUE;
		END_CASE
	END_IF

	IF xClearConifgErrStation THEN
		T_Station.TControl.xError:=FALSE;
		xClearConifgErrStation:=FALSE;
		(* Clear error station done *)
		xClearError_Done:=TRUE;
	END_IF;

	IF xClearAxis THEN
	(* Reset Error axis *)
		CASE iStepClearErrorAxis OF
		(* check station *)
		1:	xTmp:=	T_Station.THardware.TAxisToolLeft.T_CtrleSingle.xErr OR
					(T_Station.THardware.TAxisToolCenter.T_CtrleSingle.xErr AND xActiveMicroRod) OR
					T_Station.THardware.TAxisToolRight.T_CtrleSingle.xErr OR
					T_Station.THardware.TAxisToolFeeder.T_CtrleSingle.xErr OR
					T_Station.THardware.TAxisGrindFeeder.T_CtrleSingle.xErr;
			IF xTmp THEN iStepClearErrorAxis:=10;
			ELSE iStepClearErrorAxis:=90; END_IF
			iTryAgain:=0;
		(* activ clear error *)
		10:	T_Station.THardware.TAxisToolLeft.T_CtrleSingle.iFunction:=1;
			T_Station.THardware.TAxisToolLeft.T_CtrleSingle.xExecute:=T_Station.THardware.TAxisToolLeft.T_CtrleSingle.xErr;
			IF xActiveMicroRod THEN
				T_Station.THardware.TAxisToolCenter.T_CtrleSingle.iFunction:=1;
				T_Station.THardware.TAxisToolCenter.T_CtrleSingle.xExecute:=T_Station.THardware.TAxisToolCenter.T_CtrleSingle.xErr;
			END_IF;
			T_Station.THardware.TAxisToolRight.T_CtrleSingle.iFunction:=1;
			T_Station.THardware.TAxisToolRight.T_CtrleSingle.xExecute:=T_Station.THardware.TAxisToolRight.T_CtrleSingle.xErr;
			T_Station.THardware.TAxisToolFeeder.T_CtrleSingle.iFunction:=1;
			T_Station.THardware.TAxisToolFeeder.T_CtrleSingle.xExecute:=T_Station.THardware.TAxisToolFeeder.T_CtrleSingle.xErr;
			T_Station.THardware.TAxisGrindFeeder.T_CtrleSingle.iFunction:=1;
			T_Station.THardware.TAxisGrindFeeder.T_CtrleSingle.xExecute:=T_Station.THardware.TAxisGrindFeeder.T_CtrleSingle.xErr;
			(* next step *)
			iStepClearErrorAxis:=20;
			xStepClearDone:=FALSE;
		(* waiting end clearing error *)
		20:	IF NOT(xStepClearDone) THEN
			(* release action *)
				xStepClearDone:=TRUE;
			ELSE
				xTmp:=	T_Station.THardware.TAxisToolLeft.T_CtrleSingle.xDone AND
						((T_Station.THardware.TAxisToolCenter.T_CtrleSingle.xDone AND xActiveMicroRod) OR NOT(xActiveMicroRod)) AND
						T_Station.THardware.TAxisToolRight.T_CtrleSingle.xDone AND
						T_Station.THardware.TAxisToolFeeder.T_CtrleSingle.xDone AND
						T_Station.THardware.TAxisGrindFeeder.T_CtrleSingle.xDone;
				xTmp1:=	T_Station.THardware.TAxisToolLeft.T_CtrleSingle.xErr OR
						(T_Station.THardware.TAxisToolCenter.T_CtrleSingle.xErr AND xActiveMicroRod) OR
						T_Station.THardware.TAxisToolRight.T_CtrleSingle.xErr OR
						T_Station.THardware.TAxisToolFeeder.T_CtrleSingle.xErr OR
						T_Station.THardware.TAxisGrindFeeder.T_CtrleSingle.xErr;
				IF xTmp THEN
				(* confirm clear error, next step *)
					iStepClearErrorAxis:=90;
					xStepClearDone:=FALSE;
				END_IF
				IF xTmp1 THEN
					iTryAgain:=iTryAgain + 1;
					IF (iTryAgain <= 3) THEN
						(* Reset maximal three times *)
						iStepClearErrorAxis:=10;
					ELSE
						iStepClearErrorAxis:=99;
					END_IF;
				END_IF

			END_IF
		(* Clear error station done *)
		90:	xClearError_Done:=TRUE;
		(* Error *)
		99:	xClearError_Done:=TRUE;
		END_CASE;
	END_IF;

	IF xClearStandardError THEN
	(* Reset Error standard *)
		CASE iStepClearStandardError OF
		(* check NovRAM state *)
		1:	iStepClearStandardError:=10;
			IF T_NovRAM.T_Ctrle.xErr THEN T_NovRAM.T_Ctrle.xReset:=TRUE; END_IF
		(* check Profile State *)
		10:	iStepClearStandardError:=20;
			IF T_Profile.T_Ctrle.xErr THEN T_Profile.T_Ctrle.xReset:=TRUE; END_IF
		(* check HDD state *)
		20:	iStepClearStandardError:=90;
			IF T_HDD.T_Ctrle.xErr THEN T_HDD.T_Ctrle.xReset:=TRUE; END_IF
		(* Clear error station done *)
		90:	xClearError_Done:=TRUE;
		END_CASE
	END_IF

(* FB Done/Err/NotReady *)
	IF xClearError_Done OR xClearError_Err OR xClearError_NotReady THEN
	(* copy value *)
		T_Message.iState:=0;
		T_Message.sDynamicTextEnglish:='';
		T_Message.sDynamicTextDeutsch:='';
		T_Message.sDynamicTextFrancais:='';
		xDone:=xClearError_Done;
		xNotReady:=xClearError_NotReady;
		xErr:=FALSE;
		udiErrorID:=udiClearError_ErrorID;
		(* Init. function state *)
		xClearProcess:=FALSE;
		xClearStation:=FALSE;
		xClearAxis:=FALSE;
		xClearStandardError:=FALSE;
		xClearConifgErrStation:=FALSE;
	END_IF
END_FUNCTION_BLOCK

(* POU GENERAL/FB_CALCPROCESSTIME, ST *)
FUNCTION_BLOCK FB_CALCPROCESSTIME
VAR_INPUT
	T_Geometry:ST_GEOMETRY;									(* Structure of the NovRAM parameter *)
	T_AutoGeometryPara:ST_EXCHG_PARAM_AUTOGEOMETRY;		(* Structure of the NovRAM parameter *)
	T_CalibrationPara:ST_EXCHG_PARAM_CALIBRATION;			(* Structure of the NovRAM parameter *)
	T_AutoGroovePara:ST_EXCHG_PARAM_AUTOGROOVE;			(* Structure of the NovRAM parameter *)
	T_ProcessPara:ST_EXCHG_PARAM_PROCESS;					(* Structure of the NovRAM parameter *)
	rToolRotationSpeed:REAL;										(* Speed of the ToolRotation in U/Min *)
	rToolDiameter:REAL;											(* Diameter of the Tool in um *)
	rToolDiameterWithOffset:REAL;			(* diameter of the unworked Tool plus the offset for plunge and displace procedure *)
	iAutoProcess:INT;												(* 0=Calibration, 1=AutoGeometry process, 2=AutoGroove process *)
	xMicroRodActive:BOOL;										(* choice of the machine MicroWire or MicroRod *)
END_VAR
VAR_IN_OUT
	T_WorkTool:ST_WORKTOOL;									(* Tool parameter *)
END_VAR
VAR_OUTPUT
	rProcessTime: REAL;											(* calculated process time *)
END_VAR
VAR
	FBToolCalcul:FB_TOOL_CALCUL;
	ii: INT;
	rTimeLeftWork: REAL;
	iStartSection: INT;
	iEndSection: INT;
	rPlungeGrind: REAL;
	rDisplaceGrind: REAL;
	rGrindFeederPlunge: REAL;
	xResetFB: BOOL;
	xInitFB:BOOL;
(*11.10.2010 KFS {	*)
	FBCalcPlungeGrinding: FB_CALC_PLUNGE_GRINDING;
	FBCalcPlungeGrindingMultiCycle: FB_CALC_PLUNGE_GRINDING_MultiCycle;
(*11.10.2010 KFS }	*)
	rPlungeCycleGrindFeedGeometry: REAL;
	iTmpStartSection: INT;
	xCalculation: BOOL;
	rToolFeedLength: REAL;
	rSpeedToolFeed: REAL;
	rTimeAddLeftWork:REAL;
	rToolLength:REAL;
	rPlungeGrind2: REAL;
	rTimeAddLeftWorkPlungeGrind: REAL;
	rTimeAddLeftWorkPlungeGrind2: REAL;
	rTimeAddLeftWorkToolFeed: REAL;
END_VAR
(****************************************************************************************************************************************************)
(***********        This Functionblock calculates the time,  needed to work a geometry, groove or  calibration      		    ************)
(****************************************************************************************************************************************************)
	rProcessTime:=0.0;
	rTimeLeftWork:=0;
	iStartSection:=0;
	iEndSection:=0;
	xInitFB:=FALSE;
	IF (iAutoProcess = 1) THEN
	(* calculate the time for the process AutoGeometry or AutoGroove *)
		T_WorkTool.iTotalCountDownPlungeCycle:=0;
		(* Check Start and End Section of the ToolGeometry *)
		FOR ii:=1 TO 6 DO
			IF T_Geometry.axActiveSection[ii] THEN
				IF (iStartSection = 0) THEN
					iStartSection:=ii;
				END_IF;
				iEndSection:=ii;
			END_IF;
		END_FOR;
		xResetFB:=TRUE;
		(* reset first the FB for calculate the grinding plunge for each sections *)
		FBCalcPlungeGrindingMultiCycle(	rToolDiameter:= rToolDiameter,
										rToolDiameterWithOffset:=rToolDiameterWithOffset,
										xReset:= xResetFB,
										xInit:=xInitFB);
		xInitFB:=TRUE;
		FBCalcPlungeGrindingMultiCycle(	T_Geometry:= T_Geometry,
										T_AutoGeometryPara:= T_AutoGeometryPara,
										rToolDiameter:= rToolDiameter,
										rToolDiameterWithOffset:=rToolDiameterWithOffset,
										rPlungeCycleGrindFeedGeometry:=rPlungeCycleGrindFeedGeometry,
										iStartSection:= iStartSection,
										iEndSection:= iEndSection,
										xReset:= xResetFB,
										xInit:=xInitFB);

